(* Logix 5000 project; controller PBS_Perfusion vendor 1 type 14 code 217 rev 32.14; software revision 32.03; part 17 of 27 *)
(* tags used below, declared in another part *)
   P_Intlk : BOOL;   // Unique Parameter Name for auto - discovery
   REAL : DINT;
(* P_Intlk, continued *)

ROUTINE Prescan   (* ladder *)
// Clear "lurking" Commands
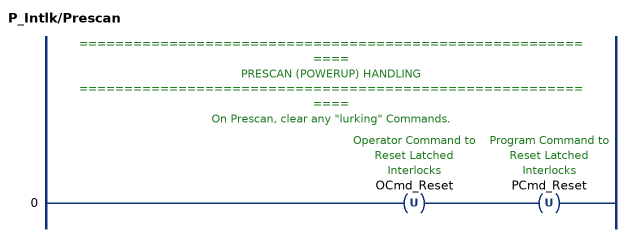
   // ============================================================
   // PRESCAN (POWERUP) HANDLING
   // ============================================================
   // On Prescan, clear any "lurking" Commands.
   0: OTU(OCmd_Reset)OTU(PCmd_Reset);
END_ROUTINE
END_ADD_ON_INSTRUCTION

ADD_ON_INSTRUCTION P_ValveC   (* revision 4.10 .01 Release, vendor Rockwell Automation, ExecutePrescan, ExecuteEnableInFalse *)
// Revision note:
// See Instruction Help for a summary of changes, and see 4.10 Release Notes for details.
// Help:
// Copyright © Rockwell Automation, Inc.  All Rights Reserved.
// This Instruction controls an Analog or Pulse Output Valve with
// analog or simulated position feedback and provides:
// *  Program and Operator entry of target position in Percent Open
// *  Ramping of position to target at specified Rate of Change (%/sec)
// *  Scaling of Position Feedback input from Raw (I/O card) Units to percent
// *  Monitoring of Interlock conditions which cause output to shed
// *  Configurable shed to HOLD or to configured position
// *  Monitoring of I/O communication faults
// *  Alarms for Interlock Trip, Actuator Fault, I/O Fault
// *  Operation in Hand, Maintenance, Override, Program and Operator Modes
// *  "Available" status for use by automation logic to know whether valve
//       can be controlled by other objects.
// Command Sources are arbitrated by a P_CmdSrc Add-On Instruction instance.
// Alarms are provided by P_Alarm Add-On Instruction instances.
// Command Sources: Operator, Program, External, Override, Maintenance, Out of Service, Hand
// Configuration notes:
//    If Max ON Time is less than 0 or greater than the Cycle Time
//         it is set to the Cycle Time.
//    If Min ON Time is less than 0 or greater than the Max ON Time
//         it is set to zero.
//    If Deadtime is less than 0 or greater than the Cycle Time,
//         it is set to zero.
//    Bump Time must be within the Min ON Time and Max ON Time.
// SUMMARY OF CHANGES FROM PREVIOUS VERSION (4.10.00)
// See 4.10 Release Notes for details.
// * No changes, uprevved because P_CmdSrc 4.10.01 is used.
// SUMMARY OF CHANGES FROM PREVIOUS VERSION (4.00.00)
// See 4.10 Release Notes for details.
// * Added option to clamp to a full/empty range when we have limit switches.
// * Changed availability to use input availability from interlocks.
// * Updated to P_CmdSrc V4.10.00.
// * Corrected parameter External Access.
// * Added Cfg_HasMoreObj.
// SUMMARY OF CHANGES FROM PREVIOUS VERSION (3.5-11)
// See 4.00 Release Notes for details.
// * Changed Inf_ items to HMI_, and added Cfg_Area for security.
// * Added notify and unack count rollup for associated object(s).
// * Changed "Mode" to "Command Source" using P_CmdSrc 4.00.00.
// * Deleted Cfg_PCmdClear; all Program Commands are now self-clearing.
// * Aligned ready bit naming with command bit names.
// * Added unacked alarm count.
// * Added  configurable decimal places for display on HMI.
// * All OCmds/MCmds and ORdys/MRdys are now Local Tags.
// * Added Sts_RdyAck and Sts_RdyReset for use by external objects.
// * Added option for no position feedback (simulated with hysteresis).
VAR_INPUT
   Inp_PosFdbk : REAL; {visible}   // Position Feedback from Valve (in Raw Input units)
   Inp_OpenLS : BOOL; {visible}   // Valve Open Limit Switch 1=confirmed fully open
   Inp_ClosedLS : BOOL; {visible}   // Valve Closed Limit Switch 1=confirmed fully closed
   Inp_ActuatorFault : BOOL; {visible}   // Valve Actuator Fault (overload, etc.), 0=OK, 1=Fault)
   Inp_IntlkOK : BOOL := 1; {visible}   // 1=Interlocks OK, Pulse Output Valve can be moved
   Inp_NBIntlkOK : BOOL := 1; {visible}   // 1=Non-Bypassable Interlocks OK, Pulse Output Valve can be moved
   Inp_IntlkAvail : BOOL;   // 1 = Interlock Availibility OK
   Inp_IOFault : BOOL;   // Input / Output Communication Status 0=OK, 1=fail
   Inp_Sim : BOOL;   // 1=I/O are being simulated, set output CV to 0.0, ignore I/O Fault
   Inp_Hand : ALIAS FOR CmdSrc.Inp_Hand;
   Inp_Ovrd : ALIAS FOR CmdSrc.Inp_Ovrd;
   Inp_OvrdCV : REAL;   // CV target in Override Mode (CV EU)
   Inp_ExtInh : ALIAS FOR CmdSrc.Inp_ExtInh;
   Inp_Reset : BOOL;   // 1=Reset shed latches and cleared alarms
   Cfg_ShedHold : BOOL;   // 1=Hold Output on Interlock or bad PV, 0=Go to Cfg_IntlkCV
   Cfg_ShedOnIOFault : BOOL := 1;   // 1=Take shed action (hold or interlock CV) on I/O Fault
   Cfg_SkipRoCLim : BOOL;   // 1=Skip RoC Limiting in Intlk, Maint, Ovrd modes
   Cfg_SetTrack : BOOL := 1;   // 1=PSets track OSets in Oper, OSets track PSets in Prog, 0=no tracking
   Cfg_SetTrackOvrdHand : BOOL;   // 1=Prog/Oper Settings track Override/Hand CV
   Cfg_HasPosFdbk : BOOL := 1;   // 1=Valve provides an analog position feedback, 0=simulate feedback
   Cfg_HasOpenLS : BOOL;   // 1=Valve provides an Open Limit Switch signal
   Cfg_HasClosedLS : BOOL;   // 1=Valve provides a Closed Limit Switch signal
   Cfg_UseOpenLS : BOOL;   // 1=Valve Open LS should be used for open/closed status
   Cfg_UseClosedLS : BOOL;   // 1=Valve Closed LS should be used for open/closed status
   Cfg_LSFail : BOOL := 1;   // 1=both switches ON=fail, 0=both switches OFF=fail
   Cfg_ClampPosToLS : BOOL;   // 1=Clamps Val_Pos to EUMin/Max when on a Limit Switch
   Cfg_HasIntlkObj : BOOL;   // 1=Tells HMI a P_Intlk is connected to Inp_Intlk
   Cfg_HasMoreObj : BOOL;   // 1=Tells HMI an object with more info is available
   Cfg_HasCVNav : BOOL;   // 1=Tells HMI to enable navigation to a connected CV object
   Cfg_OvrdIntlk : BOOL;   // 1=Override ignores Bypassable Intlk; 0=always use Intlk
   Cfg_DecPlcs : DINT;   // Number of decimal places for CV display (0..6)
   Cfg_HasIntlkTripAlm : ALIAS FOR IntlkTrip.Cfg_Exists;   // 1=Interlock Trip Alarm exists and will be checked
   Cfg_HasActuatorFaultAlm : ALIAS FOR ActuatorFault.Cfg_Exists;   // 1=Actuator Fault Alarm exists and will be checked
   Cfg_HasIOFaultAlm : ALIAS FOR IOFault.Cfg_Exists;   // 1=I/O Fault Alarm exists and will be checked
   Cfg_IntlkTripResetReqd : ALIAS FOR IntlkTrip.Cfg_ResetReqd;   // 1=Reset required to clear Interlock Trip Alarm
   Cfg_ActuatorFaultResetReqd : ALIAS FOR ActuatorFault.Cfg_ResetReqd;   // 1=Reset required to clear Actuator Fault Alarm
   Cfg_IOFaultResetReqd : ALIAS FOR IOFault.Cfg_ResetReqd;   // 1=Reset required to clear I/O Fault Alarm
   Cfg_IntlkTripAckReqd : ALIAS FOR IntlkTrip.Cfg_AckReqd;   // 1=Acknowledge required for Interlock Trip Alarm
   Cfg_ActuatorFaultAckReqd : ALIAS FOR ActuatorFault.Cfg_AckReqd;   // 1=Acknowledge required for Actuator Fault Alarm
   Cfg_IOFaultAckReqd : ALIAS FOR IOFault.Cfg_AckReqd;   // 1=Acknowledge required for I/O Fault Alarm
   Cfg_IntlkTripSeverity : ALIAS FOR IntlkTrip.Cfg_Severity;   // Interlock Trip Alarm Severity: 1..250=Low, 251..500=Medium, 501..750=High, 751..1000=Urgent
   Cfg_ActuatorFaultSeverity : ALIAS FOR ActuatorFault.Cfg_Severity;   // Actuator Fault Alarm Severity: 1..250=Low, 251..500=Medium, 501..750=High, 751..1000=Urgent
   Cfg_IOFaultSeverity : ALIAS FOR IOFault.Cfg_Severity;   // I/O Fault Alarm Severity: 1..250=Low, 251..500=Medium, 501..750=High, 751..1000=Urgent
   Cfg_MinCV : REAL;   // Minimum CV (in CV EU, for limiting)
   Cfg_MaxCV : REAL := 100.0;   // Maximum CV (in CV EU, for limiting)
   Cfg_CVRoCLimInc : REAL;   // CV Rate of Change Limit, Increasing, (EU/sec, 0=unlimited)
   Cfg_CVRoCLimDec : REAL;   // CV Rate of Change Limit, Decreasing, (EU/sec, 0=unlimited)
   Cfg_IntlkCV : REAL;   // CV (target in EU) when interlocked (if not Cfg_ShedHold)
   Cfg_CVEUMin : REAL;   // CV Minimum in Engineering Units (for scaling)
   Cfg_CVEUMax : REAL := 100.0;   // CV Maximum in Engineering Units (for scaling)
   Cfg_CVRawMin : REAL;   // CV Minimum in I/O (raw) Units (for scaling)
   Cfg_CVRawMax : REAL := 100.0;   // CV Maximum in I/O (raw) Units (for scaling)
   Cfg_FdbkRawMin : REAL;   // Position Feedback Minimum in raw input units (for scaling)
   Cfg_FdbkRawMax : REAL := 100.0;   // Position Feedback Maximum in raw input units (for scaling)
   Cfg_CycleT : REAL := 10.0;   // Open and Close Pulse Output overall period (s)
   Cfg_OpenRate : REAL := 1.0;   // Rate at which valve moves when opening (CV EU/sec)
   Cfg_CloseRate : REAL := 1.0;   // Rate at which valve moves when closing (CV EU/sec)
   Cfg_MaxOnT : REAL := 5.0;   // Open and Close Pulse Output maximum ON time (s)
   Cfg_MinOnT : REAL := 1.0;   // Open and Close Pulse Output minimum ON time (s)
   Cfg_BumpT : REAL;   // Time to bump valve open or closed (by Oper) when Fdbk Bad (sec)
   Cfg_Deadtime : REAL;   // Additional time on first pulse after stop or direction change
   Cfg_MaxClosedPos : REAL;   // Position above which valve is assumed open if limit switches not used
   PSet_CV : REAL;   // Program Setting of Controlled Variable (output) (CV EU)
   PSet_Owner : DINT;   // Program Owner Request ID (non-zero) or Release (zero)
   XSet_CV : REAL;   // External Setting of Controlled Variable (output) (CV EU)
   PCmd_Prog : ALIAS FOR CmdSrc.PCmd_Prog;
   PCmd_Oper : ALIAS FOR CmdSrc.PCmd_Oper;
   PCmd_Lock : ALIAS FOR CmdSrc.PCmd_Lock;
   PCmd_Unlock : ALIAS FOR CmdSrc.PCmd_Unlock;
   PCmd_Normal : ALIAS FOR CmdSrc.PCmd_Normal;
   PCmd_Reset : BOOL;   // Program Command to reset shed latches and cleared alarms
   PCmd_IntlkTripAck : ALIAS FOR IntlkTrip.PCmd_Ack;   // Program Command to Acknowledge Interlock Trip Alarm
   PCmd_IntlkTripSuppress : ALIAS FOR IntlkTrip.PCmd_Suppress;   // Program Command to Suppress Interlock Trip Alarm
   PCmd_IntlkTripUnsuppress : ALIAS FOR IntlkTrip.PCmd_Unsuppress;   // Program Command to Unsuppress Interlock Trip Alarm
   PCmd_IntlkTripUnshelve : ALIAS FOR IntlkTrip.PCmd_Unshelve;   // Program Command to Unshelve Interlock Trip Alarm
   PCmd_ActuatorFaultAck : ALIAS FOR ActuatorFault.PCmd_Ack;   // Program Command to Acknowledge Actuator Fault Alarm
   PCmd_ActuatorFaultSuppress : ALIAS FOR ActuatorFault.PCmd_Suppress;   // Program Command to Suppress Actuator Fault Alarm
   PCmd_ActuatorFaultUnsuppress : ALIAS FOR ActuatorFault.PCmd_Unsuppress;   // Program Command to Unsuppress Actuator Fault Alarm
   PCmd_ActuatorFaultUnshelve : ALIAS FOR ActuatorFault.PCmd_Unshelve;   // Program Command to Unshelve Actuator Fault Alarm
   PCmd_IOFaultAck : ALIAS FOR IOFault.PCmd_Ack;   // Program Command to Acknowledge I/O Fault Alarm
   PCmd_IOFaultSuppress : ALIAS FOR IOFault.PCmd_Suppress;   // Program Command to Suppress I/O Fault Alarm
   PCmd_IOFaultUnsuppress : ALIAS FOR IOFault.PCmd_Unsuppress;   // Program Command to Unsuppress I/O Fault Alarm
   PCmd_IOFaultUnshelve : ALIAS FOR IOFault.PCmd_Unshelve;   // Program Command to Unshelve I/O Fault Alarm
   MCmd_Rel : ALIAS FOR CmdSrc.MCmd_Rel;
   OCmd_Unlock : ALIAS FOR CmdSrc.OCmd_Unlock;
   XCmd_Acq : ALIAS FOR CmdSrc.XCmd_Acq;
   XCmd_Rel : ALIAS FOR CmdSrc.XCmd_Rel;
   XCmd_Reset : BOOL;   // External Command to reset shed latches and cleared alarms
END_VAR
VAR_OUTPUT
   Out_CV : REAL; {access Read Only, visible}   // CV Output in Raw (I/O Card) Units
   Out_Open : BOOL; {access Read Only, visible}   // Pulse Output to drive valve Open
   Out_Close : BOOL; {access Read Only, visible}   // Pulse Output to drive valve closed
   Val_Pos : REAL; {access Read Only, visible}   // Valve actual position from feedback (CV EU)
   Val_CVSet : REAL; {access Read Only, visible}   // Value of selected CV Setting (before rate limiting, CV EU)
   Val_CVOut : REAL; {access Read Only, visible}   // Value of CV output (after clamping and ramping) (CV EU)
   Val_CVEUMin : REAL; {access Read Only}   // Minimum of scaled range = MIN (Cfg_CVEUMin, Cfg_CVEUMax)
   Val_CVEUMax : REAL := 100.0; {access Read Only}   // Maximum of scaled range = MAX (Cfg_CVEUMin, Cfg_CVEUMax)
   SrcQ_IO : DINT; {access Read Only}   // Source and Quality of primary I/O (enumeration)
   SrcQ : DINT; {access Read Only}   // Source and Quality of primary Val/Sts (enumeration)
   Val_Fdbk : DINT; {access Read Only}   // Device Feedback 0=Moving, 1=Closed, 2=Opened, 3=Limit Switch Failure
   Val_Sts : DINT; {access Read Only}   // 0=AtTarget, 1=RampClose, 2=RampOpen, 3=Clamp@Min, 4=Clamp@Max, 5=BumpClose, 6=BumpOpen
   Val_Fault : DINT; {access Read Only}   // Device Fault Status 0=none, 32=I/OFault, 34=CfgErr
   Val_NotifyAll : DINT; {access Read Only}   // Highest Alarm prio and ack status this object + channel (enum)
   Val_UnackAlmC : DINT; {access Read Only}   // Count of Unacknowledged Alarms
   Val_Owner : DINT; {access Read Only}   // Current Object Owner ID (0=not owned)
   Sts_CVInfNaN : BOOL; {access Read Only}   // 1=Selected CV is Infinite or Not A Number (1.$, 1.#NaN)
   Sts_PosInfNaN : BOOL; {access Read Only}   // 1=Inp_PosFdbk is Infinite or Not A Number (1.$, 1.#NaN)
   Sts_BumpOpen : BOOL; {access Read Only}   // 1=Bump Open Requested or Active
   Sts_BumpClose : BOOL; {access Read Only}   // 1=Bump Close Requested or Active
   Sts_Ramping : BOOL; {access Read Only}   // 1=CV is ramping to target
   Sts_Clamped : BOOL; {access Read Only}   // 1=CV Set is clamped at CVMin or CVMax
   Sts_SkipRoCLim : BOOL; {access Read Only}   // 1=Rate of Change Limiting was skipped this scan (Maint, Ovrd, Intlk, Hand)
   Sts_Active : BOOL; {access Read Only}   // 1=CV is greater than Cfg_MaxClosedPos, show valve symbol as "opened"
   Sts_Available : BOOL; {access Read Only}   // 1=Pulse Output Valve available for control by automation (Prog)
   Sts_Bypass : BOOL; {access Read Only}   // 1=Bypassable Interlocks are Bypassed
   Sts_BypActive : BOOL; {access Read Only}   // 1=Bypassing Active (Bypassed or Maintenance)
   Sts_LSFail : BOOL; {access Read Only}   // 1=Limit Switch Overlap Failure
   Sts_NotRdy : BOOL; {access Read Only}   // 1=Device Not Ready, see detail bits for reason
   Nrdy_CfgErr : BOOL; {access Read Only}   // 1=Device Not Ready: Configuration Error
   Nrdy_Intlk : BOOL; {access Read Only}   // 1=Device Not Ready: Interlock Not OK
   Nrdy_IOFault : BOOL; {access Read Only}   // 1=Device Not Ready: I/O Fault (Shed Requires Reset)
   Nrdy_OoS : BOOL; {access Read Only}   // 1=Device Not Ready: Device is Out of Service
   Sts_MaintByp : BOOL; {access Read Only}   // 1=Device has a Maintenance Bypass function active
   Sts_AlmInh : BOOL; {access Read Only}   // 1=One or more Alarms Shelved, Disabled or Suppressed
   Sts_Err : BOOL; {access Read Only, visible}   // 1=Error in Config: see detail bits for reason
   Err_Limit : BOOL; {access Read Only}   // 1=Error in Config: CV Limits swapped
   Err_EU : BOOL; {access Read Only}   // 1=Error in Config: Scaled CV EU Min = Max
   Err_Raw : BOOL; {access Read Only}   // 1=Error in Config: Raw Output Scaling Min = Max
   Err_Fdbk : BOOL; {access Read Only}   // 1=Error in Config: Raw Feedback Scaling Min = Max
   Err_Timer : BOOL; {access Read Only}   // 1=Error in Config: Invalid Timer Preset (use 0 to 2147483)
   Err_Alarm : BOOL; {access Read Only}   // 1=Error in Config: Alarm Min On Time, Shelf Time, Severity
   Sts_Hand : ALIAS FOR CmdSrc.Sts_Hand; {access Read Only, visible}
   Sts_OoS : ALIAS FOR CmdSrc.Sts_OoS; {access Read Only, visible}
   Sts_Maint : ALIAS FOR CmdSrc.Sts_Maint; {access Read Only, visible}
   Sts_Ovrd : ALIAS FOR CmdSrc.Sts_Ovrd; {access Read Only, visible}
   Sts_Ext : ALIAS FOR CmdSrc.Sts_Ext; {access Read Only, visible}
   Sts_Prog : ALIAS FOR CmdSrc.Sts_Prog; {access Read Only, visible}
   Sts_ProgLocked : ALIAS FOR CmdSrc.Sts_ProgLocked; {access Read Only}
   Sts_Oper : ALIAS FOR CmdSrc.Sts_Oper; {access Read Only, visible}
   Sts_OperLocked : ALIAS FOR CmdSrc.Sts_OperLocked; {access Read Only}
   Sts_Normal : ALIAS FOR CmdSrc.Sts_Normal; {access Read Only}
   Sts_ExtReqInh : ALIAS FOR CmdSrc.Sts_ExtReqInh; {access Read Only}
   Sts_ProgReqInh : ALIAS FOR CmdSrc.Sts_ProgReqInh; {access Read Only}
   Sts_MAcqRcvd : ALIAS FOR CmdSrc.Sts_MAcqRcvd; {access Read Only}
   Sts_RdyReset : ALIAS FOR ORdy_Reset; {access Read Only}   // 1=A latched alarm or shed condition is ready to be reset
   Sts_RdyAck : BOOL; {access Read Only}   // 1=An alarm is ready to be acknowledged
   Sts_IntlkTrip : ALIAS FOR IntlkTrip.Inp;   // 1=Status: CV held or forced by interlock NOT OK (1-shot)
   Alm_IntlkTrip : ALIAS FOR IntlkTrip.Alm;   // 1=Alarm: CV held or forced by interlock NOT OK
   Ack_IntlkTrip : ALIAS FOR IntlkTrip.Ack;   // 1=Interlock Trip Alarm has been acknowledged
   Sts_IntlkTripDisabled : ALIAS FOR IntlkTrip.Disabled;   // 1=Interlock Trip Alarm has been Disabled by Maintenance
   Sts_IntlkTripShelved : ALIAS FOR IntlkTrip.Shelved;   // 1=Interlock Trip Alarm has been Shelved by Operator
   Sts_IntlkTripSuppressed : ALIAS FOR IntlkTrip.Suppressed;   // 1=Interlock Trip Alarm has been Suppressed by Program
   Sts_ActuatorFault : ALIAS FOR ActuatorFault.Inp;   // 1=Actuator Fault detected (input)
   Alm_ActuatorFault : ALIAS FOR ActuatorFault.Alm;   // 1=Alarm: Actuator Fault Detected
   Ack_ActuatorFault : ALIAS FOR ActuatorFault.Ack;   // 1=Actuator Fault Alarm has been acknowledged
   Sts_ActuatorFaultDisabled : ALIAS FOR ActuatorFault.Disabled;   // 1=Actuator Fault Alarm has been Disabled by Maintenance
   Sts_ActuatorFaultShelved : ALIAS FOR ActuatorFault.Shelved;   // 1=Actuator Fault Alarm has been Shelved by Operator
   Sts_ActuatorFaultSuppressed : ALIAS FOR ActuatorFault.Suppressed;   // 1=Actuator Fault Alarm has been Suppressed by Program
   Sts_IOFault : ALIAS FOR IOFault.Inp;   // 1=I/O Fault Status (0=OK, 1=Bad)
   Alm_IOFault : ALIAS FOR IOFault.Alm;   // 1=I/O Fault Alarm
   Ack_IOFault : ALIAS FOR IOFault.Ack;   // 1=I/O Fault Alarm has been acknowledged
   Sts_IOFaultDisabled : ALIAS FOR IOFault.Disabled;   // 1=I/O Fault Alarm has been Disabled by Maintenance
   Sts_IOFaultShelved : ALIAS FOR IOFault.Shelved;   // 1=I/O Fault Alarm has been Shelved by Operator
   Sts_IOFaultSuppressed : ALIAS FOR IOFault.Suppressed;   // 1=I/O Fault Alarm has been Suppressed by Program
   MRdy_Rel : ALIAS FOR CmdSrc.MRdy_Rel; {access Read Only}
   ORdy_Unlock : ALIAS FOR CmdSrc.ORdy_Unlock; {access Read Only}
   P_ValveC : BOOL;   // Unique Parameter Name for auto - discovery
END_VAR
VAR
   CmdSrc : P_CmdSrc := (Cfg_HasOper := 1, Cfg_HasOperLocked := 1, Cfg_HasProg := 1, Cfg_HasProgLocked := 1, Cfg_HasMaint := 1, Cfg_HasMOoS := 1, Cfg_OvrdOverLock := 1, Sts_bSrc := 1);   // Control / Command Source Selection
   IOFault : P_Alarm := (Cfg_AckReqd := 1, Cfg_AllowShelve := 1, Cfg_AllowDisable := 1, Cfg_Severity := 1000, Cfg_AlmMinOnT := 5, PCfg_AllowExist := 1, Ack := 1);   // I/O Fault Alarm
   IntlkTrip : P_Alarm := (Cfg_AckReqd := 1, Cfg_AllowShelve := 1, Cfg_AllowDisable := 1, Cfg_Severity := 500, Cfg_AlmMinOnT := 5, PCfg_AllowExist := 1, Ack := 1);   // Interlock Trip Alarm
   Cfg_Tag : STRING_20 := 'P_ValveC';   // Tagname for display on HMI
   Cfg_Label : STRING_20 := 'Control Valve';   // Label for graphic symbol displayed on HMI
   Cfg_Desc : STRING_40 := 'Control Valve';   // Description for display on HMI
   Wrk_Notify : DINT; {access None}   // Buffer for building Val_Notify
   Wrk_Bypass : BOOL; {access None}   // Internal Bypassable Interlocks are Bypassed flag
   Cfg_EU : STRING_8 := '% Open';   // Engineering Units for display on HMI
   Wrk_CV : REAL; {access None}   // Working copy of Speed Reference (for limiting)
   Wrk_CVSet : REAL; {access None}   // Final selected CV to feed to RoC Limiter
   Wrk_CVOut : REAL; {access None}   // Working value of CV after Rate Limiting
   Wrk_IntlkTripONS : BOOL; {access None}   // Interlock Tripped This Scan
   Wrk_ScanTime : REAL; {access None}   // Seconds since previous scan
   Wrk_StepInc : REAL; {access None}   // Amount to increase CV (to valve pulse logic) this scan for rate limiting
   Wrk_ScanT : TIMER := (PRE := 2147483647); {access None}   // Scan Timer (milliseconds, always runs)
   HMI_Tab : SINT;   // Tab to display (FTView ME)
   Wrk_Sts : DINT; {access None}   // Buffer for building Val_Sts
   Wrk_Fault : DINT; {access None}   // Buffer for building Val_Fault
   Wrk_SrcQ : DINT; {access None}   // Register for building Source / Quality enumeration
   ActuatorFault : P_Alarm := (Cfg_AckReqd := 1, Cfg_AllowShelve := 1, Cfg_AllowDisable := 1, Cfg_Severity := 1000, Cfg_AlmMinOnT := 5, PCfg_AllowExist := 1, Ack := 1);   // Actuator Fault Alarm (based on Actuator Fault Input)
   Wrk_RealChkDINT : DINT; {access None}   // REAL tag bit pattern as a DINT to check for Inf / NaN
   Wrk_Close : BOOL; {access None}   // Internal Close output -- before Sim
   Wrk_Open : BOOL; {access None}   // Internal Open output -- before Sim
   Wrk_CycleT : TIMER := (PRE := 2147483647); {access None}   // Overall Cycle Timer for pulsed outputs
   Wrk_OKtoOpen : BOOL; {access None}   // OK to pulse Out_Open
   Wrk_OKtoClose : BOOL; {access None}   // OK to pulse Out_Close
   Wrk_OpenTime : REAL; {access None}   // Time to pulse Out_Open
   Wrk_CycleT_ms : DINT; {access None}   // Cycle Time in milliseconds (preset)
   Wrk_OpenTimePrev : DINT; {access None}   // Wrk_OpenTime from previous cycle
   Wrk_CloseTime : REAL; {access None}   // Time to pulse Out_Close
   Wrk_CloseTimePrev : REAL; {access None}   // Wrk_CloseTime from previous cycle
   HMI_Type : STRING_16 := 'P_ValveC'; {access Read Only}   // Must contain AOI name, used for HMI and Information S/W
   Wrk_OpenFdbk : BOOL; {access None}   // 1=LS Feedback shows valve confirmed open
   Wrk_ClosedFdbk : BOOL; {access None}   // 1=LS Feedback shows valve confirmed closed
   Wrk_StepDec : REAL; {access None}   // Amount to decrease CV (to valve pulse logic) this scan for rate limiting
   Wrk_BumpClose : BOOL; {access None}   // Operator Bump Close requested
   Wrk_BumpOpen : BOOL; {access None}   // Operator Bump Open requested
   Wrk_BumpingOpen : BOOL; {access None}   // Operator Bump Open actively pulsing Out_Open
   Wrk_BumpingClose : BOOL; {access None}   // Operator Bump Close actively pulsing Out_Close
   Wrk_CycleActive : BOOL; {access None}   // Outputs are cycling; wait for cycle to complete
   HMI_Lib : STRING_12 := 'RA-BAS'; {access Read Only}   // Display Library for Faceplate call-up
   Cfg_CVNavTag : STRING_NavTag;   // Tagname for destination of CV Navigation button
   Wrk_ShedIntlkCV : BOOL; {access None}   // Output CV being held at Interlock value
   Wrk_ShedHold : BOOL; {access None}   // Output CV being held at last good value
   Cfg_Area : STRING_Area := 'area01';   // Process Area for security
   OSet_CV : REAL;   // Operator Setting of Controlled Variable (output) (CV EU)
   OCmd_ResetAckAll : BOOL;   // Oper Cmd to reset shed latches and cleared alarms and acknowledge all alarms
   OCmd_Reset : BOOL;   // Oper Cmd to reset shed latches and cleared alarms
   MCmd_Check : BOOL;   // Maintenance Command to Check (not bypass) all Interlocks
   MCmd_Bypass : BOOL;   // Maintenance Command to Bypass all Bypassable Interlocks
   OCmd_BumpClose : BOOL;   // Operator Command to bump valve closed (avail. if Fdbk Bad)
   OCmd_BumpOpen : BOOL;   // Operator Command to bump valve open (avail. if Fdbk Bad)
   ORdy_CV : BOOL; {access Read Only}   // 1=Ready for OSet_CV (enables data entry field)
   ORdy_ResetAckAll : BOOL; {access Read Only}   // 1=Ready for OCmd_ResetAckAll (enables HMI button)
   ORdy_Reset : BOOL; {access Read Only}   // 1=Ready for OCmd_Reset (enables HMI button)
   MRdy_Check : BOOL; {access Read Only}   // 1=Ready for MCmd_Check (enables HMI button)
   MRdy_Bypass : BOOL; {access Read Only}   // 1=Ready for MCmd_Bypass (enables HMI button)
   ORdy_BumpClose : BOOL; {access Read Only}   // 1=Ready for OCmd_BumpClose (enables HMI button)
   ORdy_BumpOpen : BOOL; {access Read Only}   // 1=Ready for OCmd_BumpOpen (enables HMI button)
   Wrk_UnackAlmC : DINT; {access None}   // Buffer for building Val_UnackAlmC
   Val_Notify : DINT; {access Read Only}   // Current Alarm Level and Acknowledgement (enumeration)
   Wrk_DeadtimeT : TIMER; {access None}   // Timer for valve hysteresis (deadtime)
   Wrk_LastMove : BOOL; {access None}   // 1=Last move was to open, 0=Last move was to close
   Wrk_WaitDeadtime : BOOL; {access None}   // 1=Need to wait deadtime before simulated move
END_VAR

ROUTINE EnableInFalse   (* ladder *)
// Out of Service is asserted, Output OFF (zero), Alarms inhibited
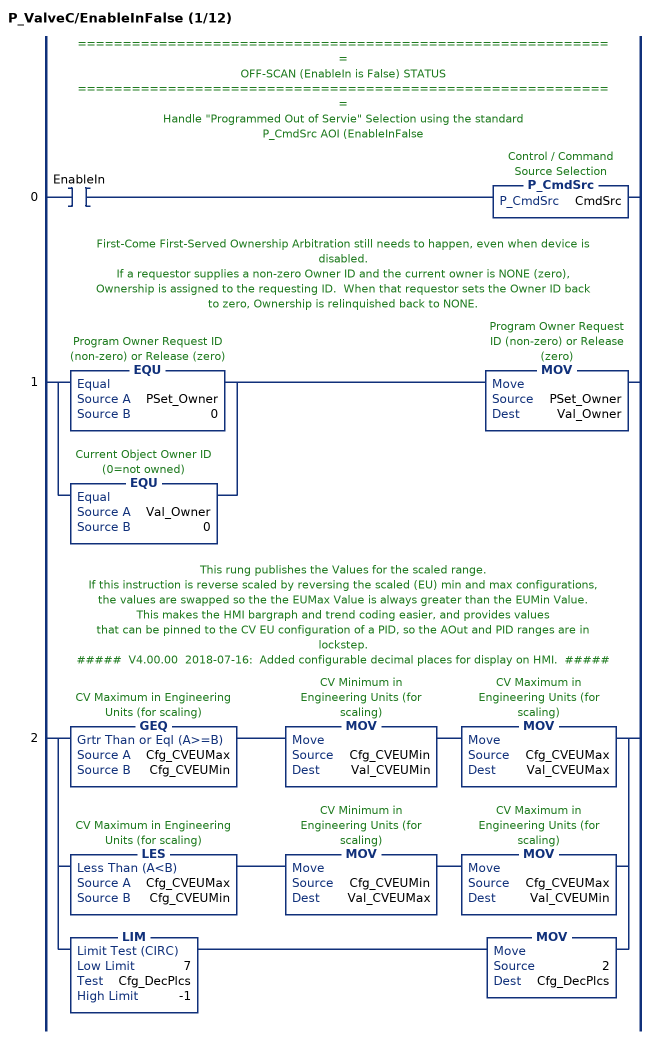
   // ============================================================
   // OFF-SCAN (EnableIn is False) STATUS
   // ============================================================
   // Handle "Programmed Out of Servie" Selection using the standard
   // P_CmdSrc AOI (EnableInFalse
   0: XIC(EnableIn)P_CmdSrc(CmdSrc);
   // First-Come First-Served Ownership Arbitration still needs to happen, even when device is disabled.
   // If a requestor supplies a non-zero Owner ID and the current owner is NONE (zero),
   // Ownership is assigned to the requesting ID.  When that requestor sets the Owner ID back
   // to zero, Ownership is relinquished back to NONE.
   1: [EQU(PSet_Owner,0) ,EQU(Val_Owner,0) ]MOV(PSet_Owner,Val_Owner);
   // This rung publishes the Values for the scaled range.
   // If this instruction is reverse scaled by reversing the scaled (EU) min and max configurations,
   // the values are swapped so the the EUMax Value is always greater than the EUMin Value.
   // This makes the HMI bargraph and trend coding easier, and provides values
   // that can be pinned to the CV EU configuration of a PID, so the AOut and PID ranges are in lockstep.
   // #####  V4.00.00  2018-07-16:  Added configurable decimal places for display on HMI.  #####
   2: [GEQ(Cfg_CVEUMax,Cfg_CVEUMin) MOV(Cfg_CVEUMin,Val_CVEUMin) MOV(Cfg_CVEUMax,Val_CVEUMax) ,LES(Cfg_CVEUMax,Cfg_CVEUMin) MOV(Cfg_CVEUMin,Val_CVEUMax) MOV(Cfg_CVEUMax,Val_CVEUMin) ,LIM(7,Cfg_DecPlcs,-1) MOV(2,Cfg_DecPlcs) ];
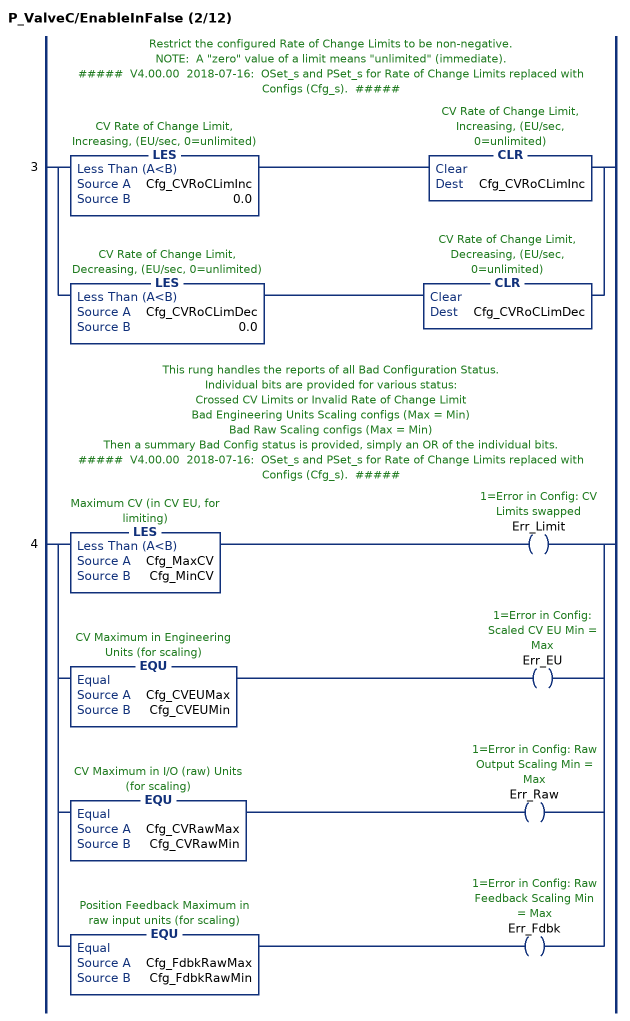
   // Restrict the configured Rate of Change Limits to be non-negative.
   // NOTE:  A "zero" value of a limit means "unlimited" (immediate).
   // #####  V4.00.00  2018-07-16:  OSet_s and PSet_s for Rate of Change Limits replaced with Configs (Cfg_s).  #####
   3: [LES(Cfg_CVRoCLimInc,0.0) CLR(Cfg_CVRoCLimInc) ,LES(Cfg_CVRoCLimDec,0.0) CLR(Cfg_CVRoCLimDec) ];
   // This rung handles the reports of all Bad Configuration Status.
   // Individual bits are provided for various status:
   // Crossed CV Limits or Invalid Rate of Change Limit
   // Bad Engineering Units Scaling configs (Max = Min)
   // Bad Raw Scaling configs (Max = Min)
   // Then a summary Bad Config status is provided, simply an OR of the individual bits.
   // #####  V4.00.00  2018-07-16:  OSet_s and PSet_s for Rate of Change Limits replaced with Configs (Cfg_s).  #####
   4: [LES(Cfg_MaxCV,Cfg_MinCV) OTE(Err_Limit) ,EQU(Cfg_CVEUMax,Cfg_CVEUMin) OTE(Err_EU) ,EQU(Cfg_CVRawMax,Cfg_CVRawMin) OTE(Err_Raw) ,EQU(Cfg_FdbkRawMax,Cfg_FdbkRawMin) OTE(Err_Fdbk) ];
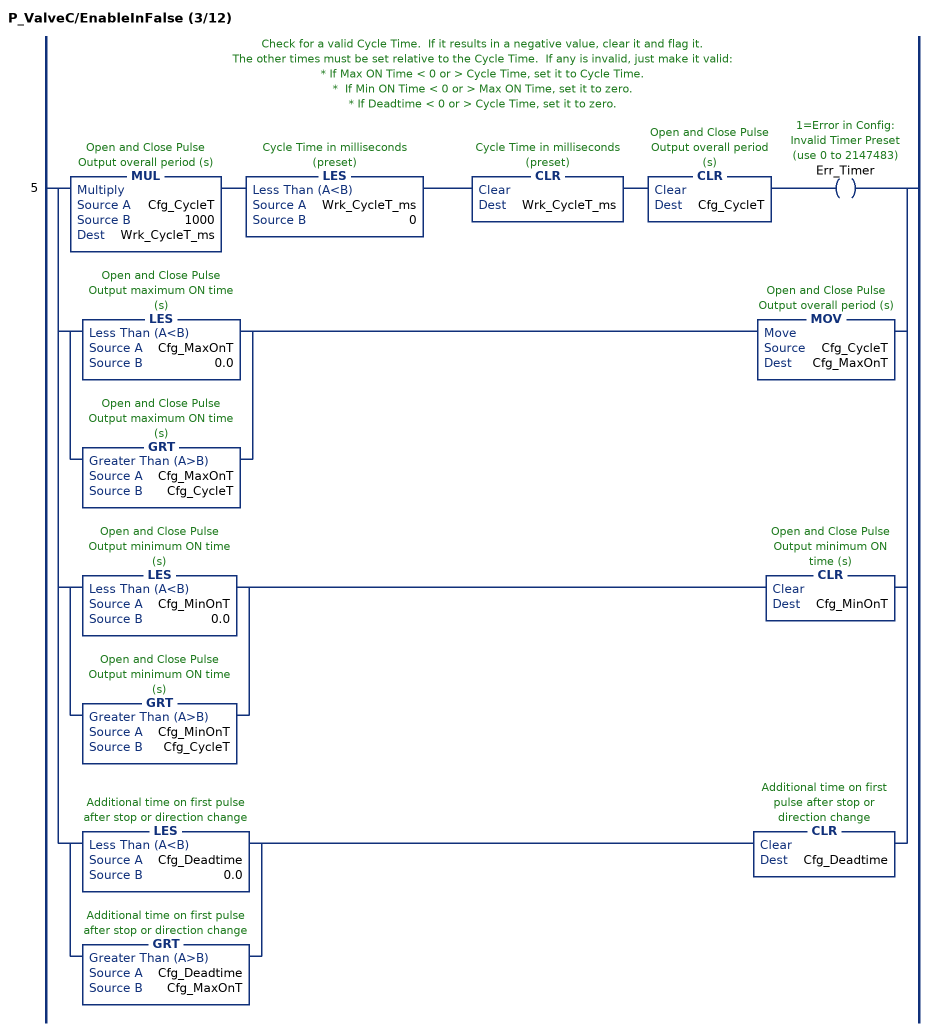
   // Check for a valid Cycle Time.  If it results in a negative value, clear it and flag it.
   // The other times must be set relative to the Cycle Time.  If any is invalid, just make it valid:
   // * If Max ON Time < 0 or > Cycle Time, set it to Cycle Time.
   // *  If Min ON Time < 0 or > Max ON Time, set it to zero.
   // * If Deadtime < 0 or > Cycle Time, set it to zero.
   5: [MUL(Cfg_CycleT,1000,Wrk_CycleT_ms) LES(Wrk_CycleT_ms,0) CLR(Wrk_CycleT_ms) CLR(Cfg_CycleT) OTE(Err_Timer) ,[LES(Cfg_MaxOnT,0.0) ,GRT(Cfg_MaxOnT,Cfg_CycleT) ] MOV(Cfg_CycleT,Cfg_MaxOnT) ,[LES(Cfg_MinOnT,0.0) ,GRT(Cfg_MinOnT,Cfg_CycleT) ] CLR(Cfg_MinOnT) ,[LES(Cfg_Deadtime,0.0) ,GRT(Cfg_Deadtime,Cfg_MaxOnT) ] CLR(Cfg_Deadtime) ];
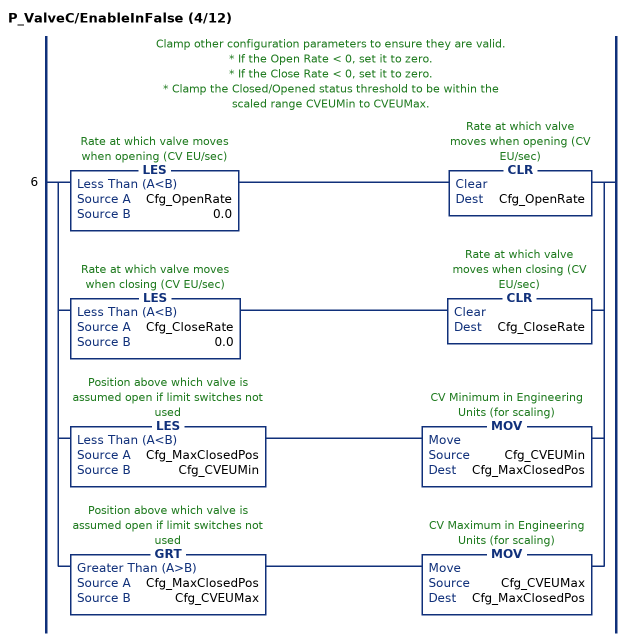
   // Clamp other configuration parameters to ensure they are valid.
   // * If the Open Rate < 0, set it to zero.
   // * If the Close Rate < 0, set it to zero.
   // * Clamp the Closed/Opened status threshold to be within the
   // scaled range CVEUMin to CVEUMax.
   6: [LES(Cfg_OpenRate,0.0) CLR(Cfg_OpenRate) ,LES(Cfg_CloseRate,0.0) CLR(Cfg_CloseRate) ,LES(Cfg_MaxClosedPos,Cfg_CVEUMin) MOV(Cfg_CVEUMin,Cfg_MaxClosedPos) ,GRT(Cfg_MaxClosedPos,Cfg_CVEUMax) MOV(Cfg_CVEUMax,Cfg_MaxClosedPos) ];
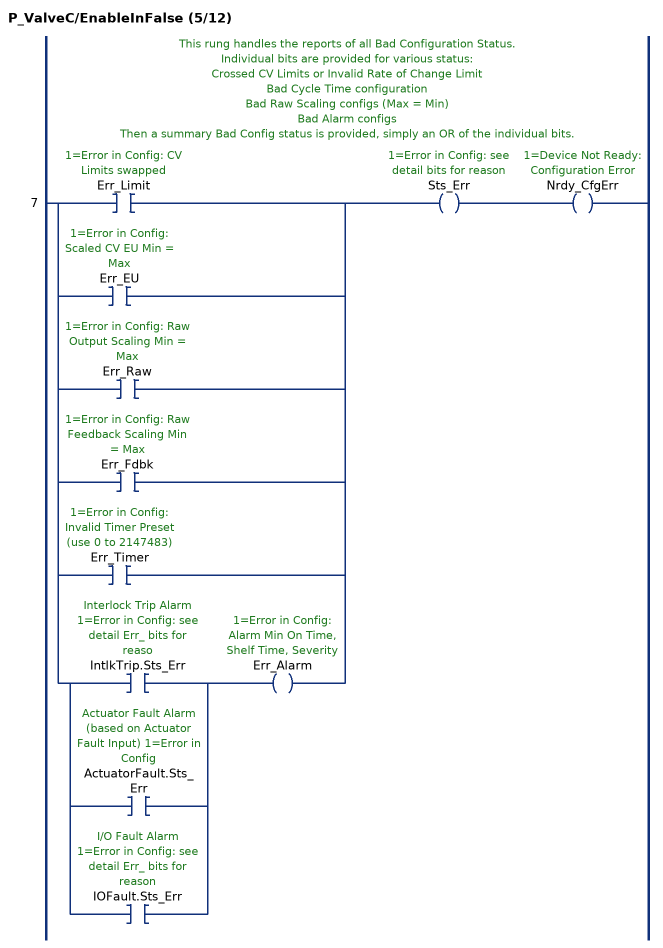
   // This rung handles the reports of all Bad Configuration Status.
   // Individual bits are provided for various status:
   // Crossed CV Limits or Invalid Rate of Change Limit
   // Bad Cycle Time configuration
   // Bad Raw Scaling configs (Max = Min)
   // Bad Alarm configs
   // Then a summary Bad Config status is provided, simply an OR of the individual bits.
   7: [XIC(Err_Limit) ,XIC(Err_EU) ,XIC(Err_Raw) ,XIC(Err_Fdbk) ,XIC(Err_Timer) ,[XIC(IntlkTrip.Sts_Err) ,XIC(ActuatorFault.Sts_Err) ,XIC(IOFault.Sts_Err) ] OTE(Err_Alarm) ]OTE(Sts_Err)OTE(Nrdy_CfgErr);
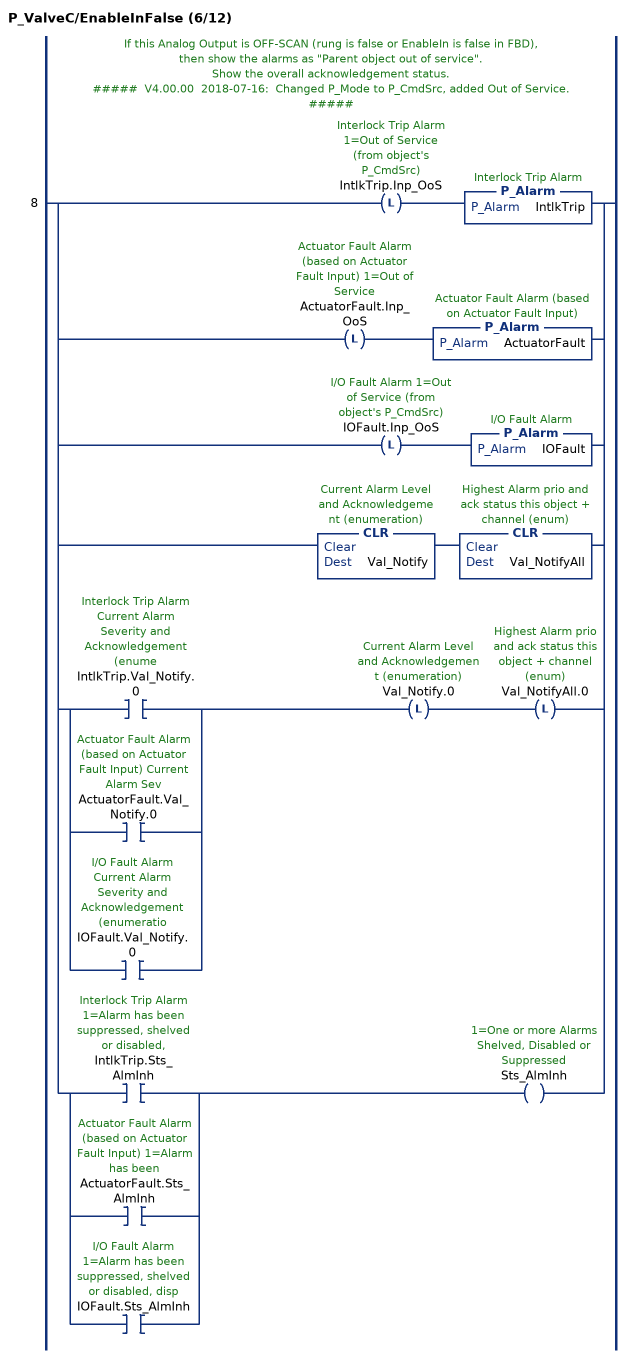
   // If this Analog Output is OFF-SCAN (rung is false or EnableIn is false in FBD),
   // then show the alarms as "Parent object out of service".
   // Show the overall acknowledgement status.
   // #####  V4.00.00  2018-07-16:  Changed P_Mode to P_CmdSrc, added Out of Service.  #####
   8: [OTL(IntlkTrip.Inp_OoS) P_Alarm(IntlkTrip) ,OTL(ActuatorFault.Inp_OoS) P_Alarm(ActuatorFault) ,OTL(IOFault.Inp_OoS) P_Alarm(IOFault) ,CLR(Val_Notify) CLR(Val_NotifyAll) ,[XIC(IntlkTrip.Val_Notify.0) ,XIC(ActuatorFault.Val_Notify.0) ,XIC(IOFault.Val_Notify.0) ] OTL(Val_Notify.0) OTL(Val_NotifyAll.0) ,[XIC(IntlkTrip.Sts_AlmInh) ,XIC(ActuatorFault.Sts_AlmInh) ,XIC(IOFault.Sts_AlmInh) ] OTE(Sts_AlmInh) ];
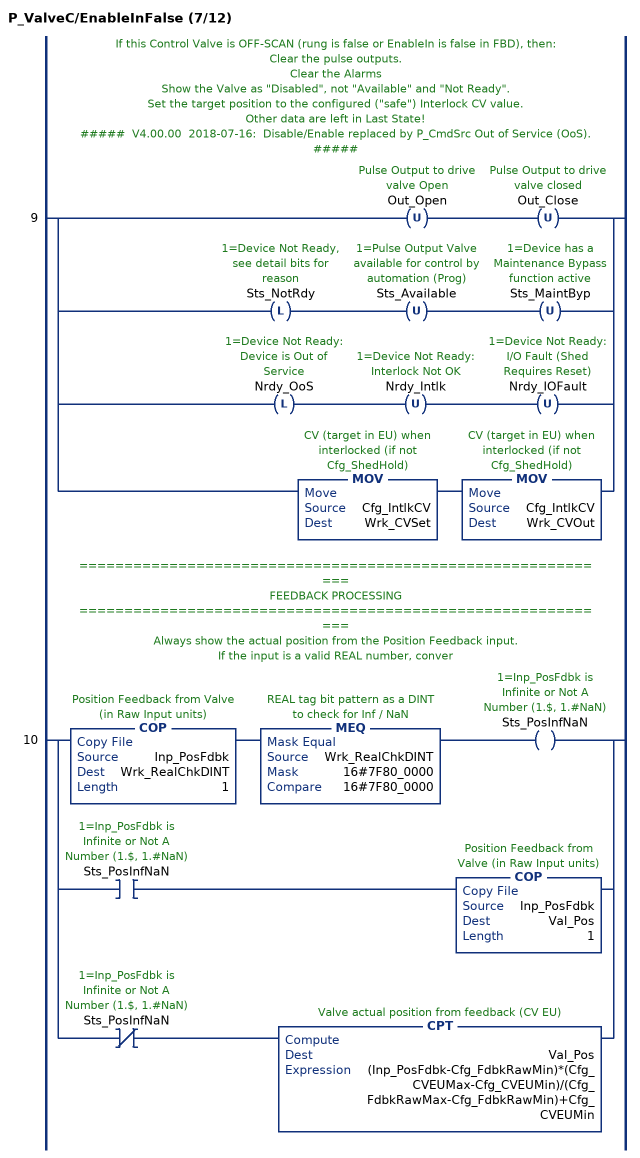
   // If this Control Valve is OFF-SCAN (rung is false or EnableIn is false in FBD), then:
   // Clear the pulse outputs.
   // Clear the Alarms
   // Show the Valve as "Disabled", not "Available" and "Not Ready".
   // Set the target position to the configured ("safe") Interlock CV value.
   // Other data are left in Last State!
   // #####  V4.00.00  2018-07-16:  Disable/Enable replaced by P_CmdSrc Out of Service (OoS).  #####
   9: [OTU(Out_Open) OTU(Out_Close) ,OTL(Sts_NotRdy) OTU(Sts_Available) OTU(Sts_MaintByp) ,OTL(Nrdy_OoS) OTU(Nrdy_Intlk) OTU(Nrdy_IOFault) ,MOV(Cfg_IntlkCV,Wrk_CVSet) MOV(Cfg_IntlkCV,Wrk_CVOut) ];
   // ============================================================
   // FEEDBACK PROCESSING
   // ============================================================
   // Always show the actual position from the Position Feedback input.
   // If the input is a valid REAL number, conver
   10: [COP(Inp_PosFdbk,Wrk_RealChkDINT,1) MEQ(Wrk_RealChkDINT,16#7F80_0000,16#7F80_0000) OTE(Sts_PosInfNaN) ,XIC(Sts_PosInfNaN) COP(Inp_PosFdbk,Val_Pos,1) ,XIO(Sts_PosInfNaN) CPT(Val_Pos,(Inp_PosFdbk-Cfg_FdbkRawMin)*(Cfg_CVEUMax-Cfg_CVEUMin)/(Cfg_FdbkRawMax-Cfg_FdbkRawMin)+Cfg_CVEUMin) ];
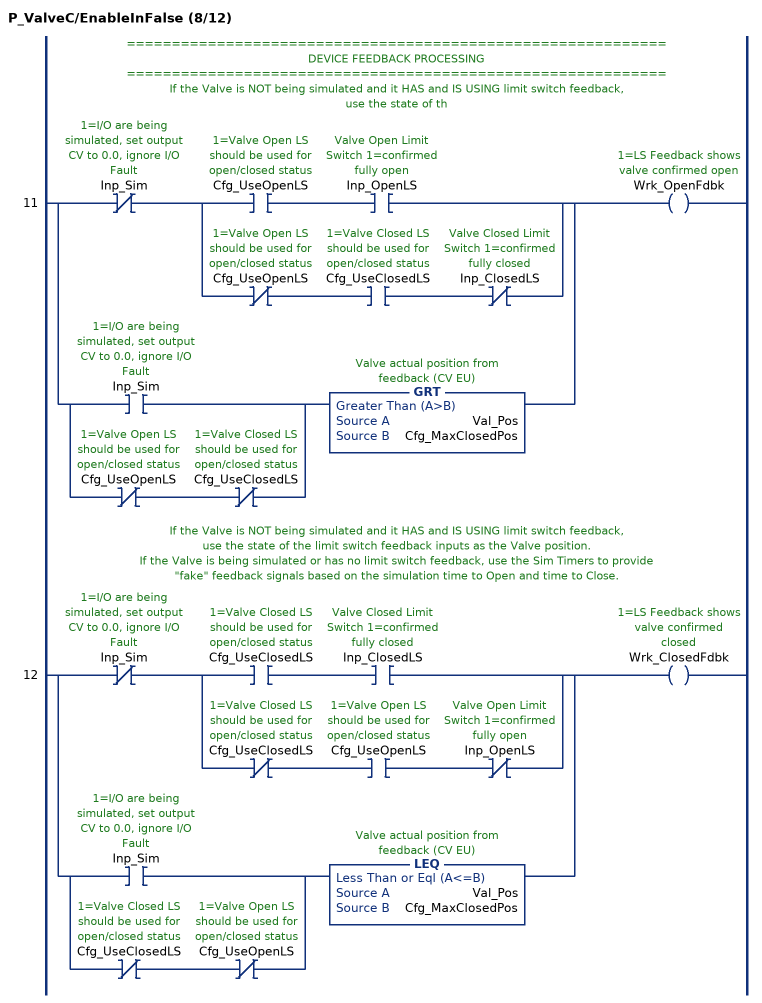
   // ============================================================
   // DEVICE FEEDBACK PROCESSING
   // ============================================================
   // If the Valve is NOT being simulated and it HAS and IS USING limit switch feedback,
   // use the state of th
   11: [XIO(Inp_Sim) [XIC(Cfg_UseOpenLS) XIC(Inp_OpenLS) ,XIO(Cfg_UseOpenLS) XIC(Cfg_UseClosedLS) XIO(Inp_ClosedLS) ] ,[XIC(Inp_Sim) ,XIO(Cfg_UseOpenLS) XIO(Cfg_UseClosedLS) ] GRT(Val_Pos,Cfg_MaxClosedPos) ]OTE(Wrk_OpenFdbk);
   // If the Valve is NOT being simulated and it HAS and IS USING limit switch feedback,
   // use the state of the limit switch feedback inputs as the Valve position.
   // If the Valve is being simulated or has no limit switch feedback, use the Sim Timers to provide
   // "fake" feedback signals based on the simulation time to Open and time to Close.
   12: [XIO(Inp_Sim) [XIC(Cfg_UseClosedLS) XIC(Inp_ClosedLS) ,XIO(Cfg_UseClosedLS) XIC(Cfg_UseOpenLS) XIO(Inp_OpenLS) ] ,[XIC(Inp_Sim) ,XIO(Cfg_UseClosedLS) XIO(Cfg_UseOpenLS) ] LEQ(Val_Pos,Cfg_MaxClosedPos) ]OTE(Wrk_ClosedFdbk);
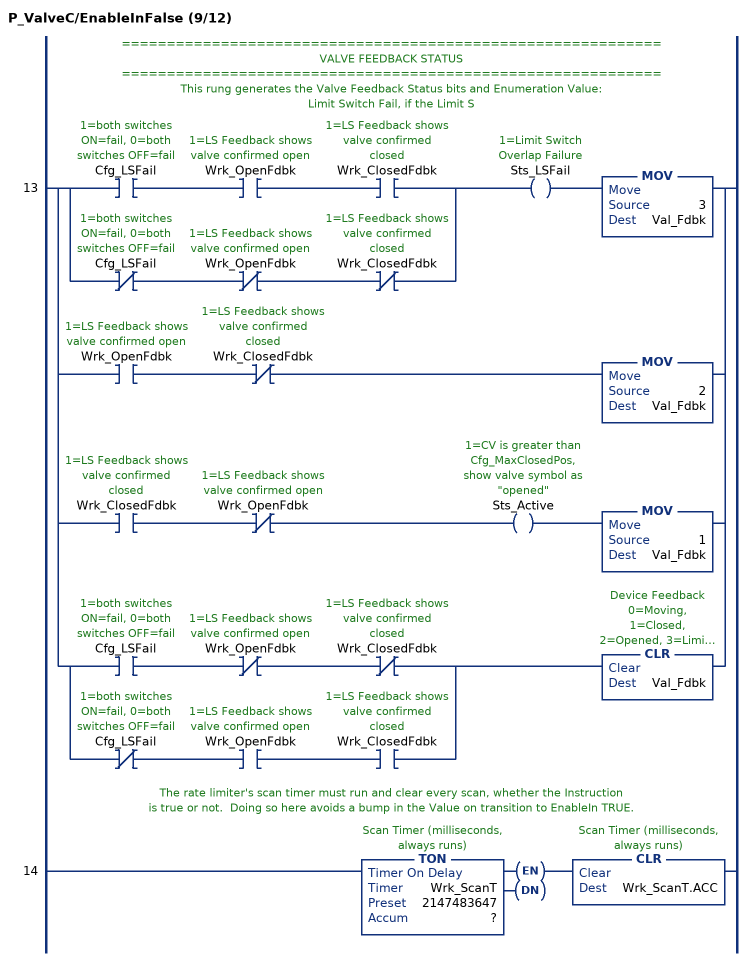
   // ============================================================
   // VALVE FEEDBACK STATUS
   // ============================================================
   // This rung generates the Valve Feedback Status bits and Enumeration Value:
   // Limit Switch Fail, if the Limit S
   13: [[XIC(Cfg_LSFail) XIC(Wrk_OpenFdbk) XIC(Wrk_ClosedFdbk) ,XIO(Cfg_LSFail) XIO(Wrk_OpenFdbk) XIO(Wrk_ClosedFdbk) ] OTE(Sts_LSFail) MOV(3,Val_Fdbk) ,XIC(Wrk_OpenFdbk) XIO(Wrk_ClosedFdbk) MOV(2,Val_Fdbk) ,XIC(Wrk_ClosedFdbk) XIO(Wrk_OpenFdbk) OTE(Sts_Active) MOV(1,Val_Fdbk) ,[XIC(Cfg_LSFail) XIO(Wrk_OpenFdbk) XIO(Wrk_ClosedFdbk) ,XIO(Cfg_LSFail) XIC(Wrk_OpenFdbk) XIC(Wrk_ClosedFdbk) ] CLR(Val_Fdbk) ];
   // The rate limiter's scan timer must run and clear every scan, whether the Instruction
   // is true or not.  Doing so here avoids a bump in the Value on transition to EnableIn TRUE.
   14: TON(Wrk_ScanT,?,?)CLR(Wrk_ScanT.ACC);
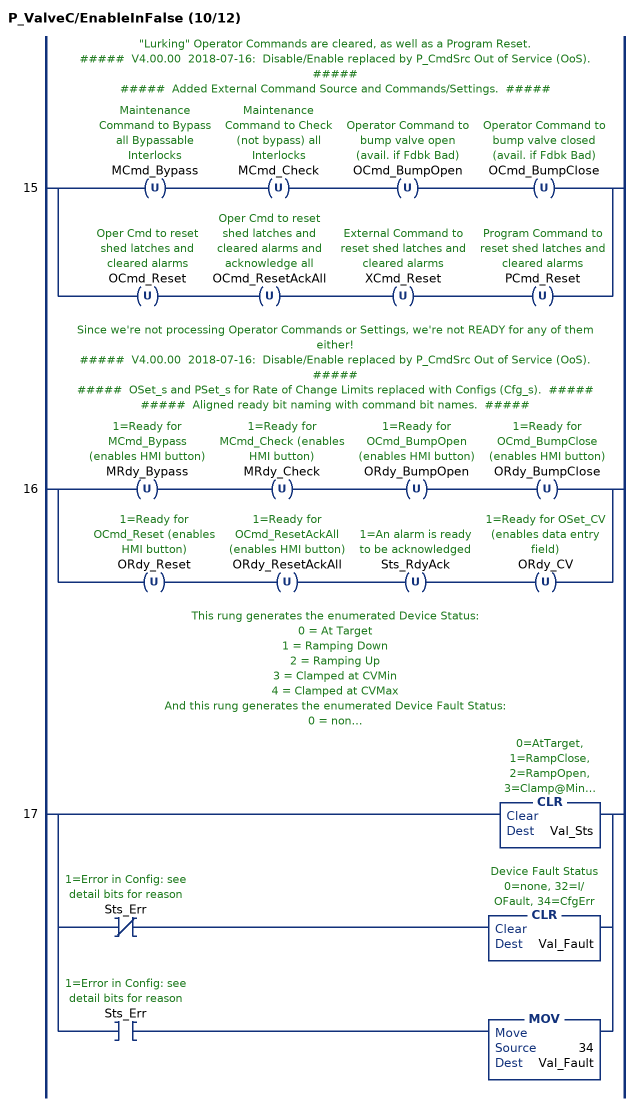
   // "Lurking" Operator Commands are cleared, as well as a Program Reset.
   // #####  V4.00.00  2018-07-16:  Disable/Enable replaced by P_CmdSrc Out of Service (OoS).  #####
   // #####  Added External Command Source and Commands/Settings.  #####
   15: [OTU(MCmd_Bypass) OTU(MCmd_Check) OTU(OCmd_BumpOpen) OTU(OCmd_BumpClose) ,OTU(OCmd_Reset) OTU(OCmd_ResetAckAll) OTU(XCmd_Reset) OTU(PCmd_Reset) ];
   // Since we're not processing Operator Commands or Settings, we're not READY for any of them either!
   // #####  V4.00.00  2018-07-16:  Disable/Enable replaced by P_CmdSrc Out of Service (OoS).  #####
   // #####  OSet_s and PSet_s for Rate of Change Limits replaced with Configs (Cfg_s).  #####
   // #####  Aligned ready bit naming with command bit names.  #####
   16: [OTU(MRdy_Bypass) OTU(MRdy_Check) OTU(ORdy_BumpOpen) OTU(ORdy_BumpClose) ,OTU(ORdy_Reset) OTU(ORdy_ResetAckAll) OTU(Sts_RdyAck) OTU(ORdy_CV) ];
   // This rung generates the enumerated Device Status:
   // 0 = At Target
   // 1 = Ramping Down
   // 2 = Ramping Up
   // 3 = Clamped at CVMin
   // 4 = Clamped at CVMax
   // And this rung generates the enumerated Device Fault Status:
   // 0 = none
   // 32 = I/O Fault
   // 34 = Configuration Error
   17: [CLR(Val_Sts) ,XIO(Sts_Err) CLR(Val_Fault) ,XIC(Sts_Err) MOV(34,Val_Fault) ];
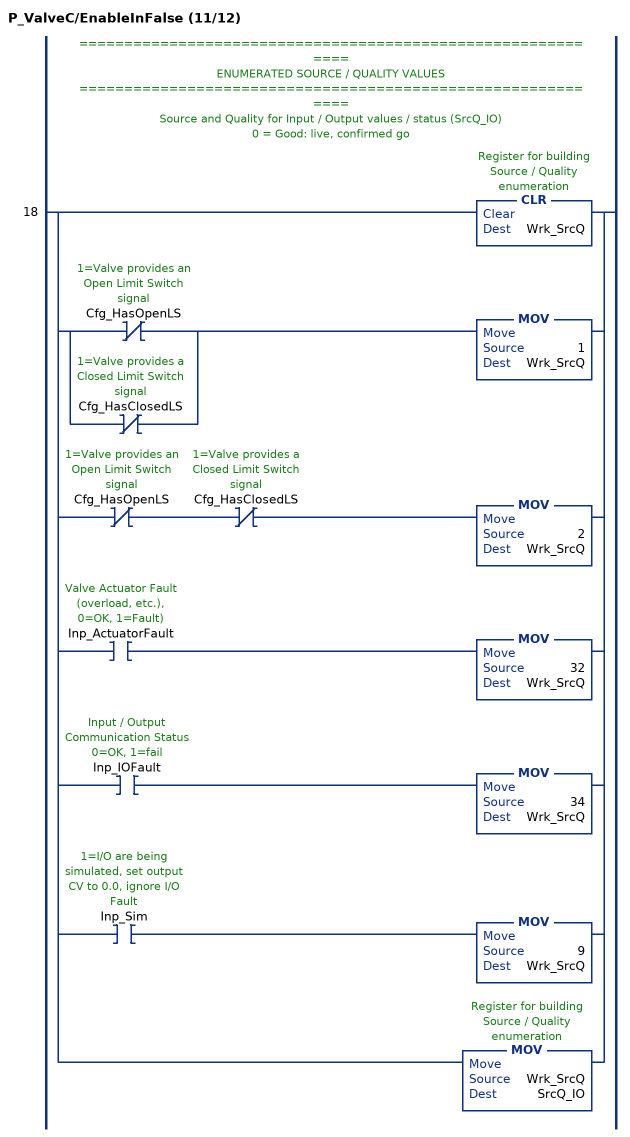
   // ============================================================
   // ENUMERATED SOURCE / QUALITY VALUES
   // ============================================================
   // Source and Quality for Input / Output values / status (SrcQ_IO)
   // 0 = Good: live, confirmed go
   18: [CLR(Wrk_SrcQ) ,[XIO(Cfg_HasOpenLS) ,XIO(Cfg_HasClosedLS) ] MOV(1,Wrk_SrcQ) ,XIO(Cfg_HasOpenLS) XIO(Cfg_HasClosedLS) MOV(2,Wrk_SrcQ) ,XIC(Inp_ActuatorFault) MOV(32,Wrk_SrcQ) ,XIC(Inp_IOFault) MOV(34,Wrk_SrcQ) ,XIC(Inp_Sim) MOV(9,Wrk_SrcQ) ,MOV(Wrk_SrcQ,SrcQ_IO) ];
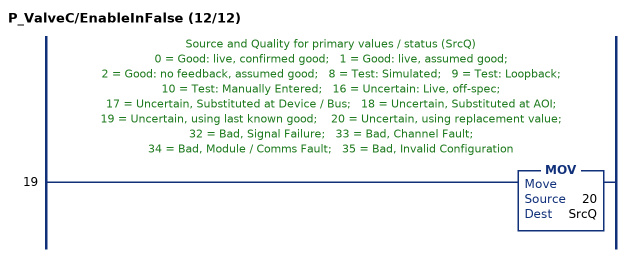
   // Source and Quality for primary values / status (SrcQ)
   // 0 = Good: live, confirmed good;   1 = Good: live, assumed good;
   // 2 = Good: no feedback, assumed good;   8 = Test: Simulated;   9 = Test: Loopback;
   // 10 = Test: Manually Entered;   16 = Uncertain: Live, off-spec;
   // 17 = Uncertain, Substituted at Device / Bus;   18 = Uncertain, Substituted at AOI;
   // 19 = Uncertain, using last known good;    20 = Uncertain, using replacement value;
   // 32 = Bad, Signal Failure;   33 = Bad, Channel Fault;
   // 34 = Bad, Module / Comms Fault;   35 = Bad, Invalid Configuration
   19: MOV(20,SrcQ);
END_ROUTINE

ROUTINE Logic   (* ladder *)
// Normal Scan: manipulate Control Valve with position feedback
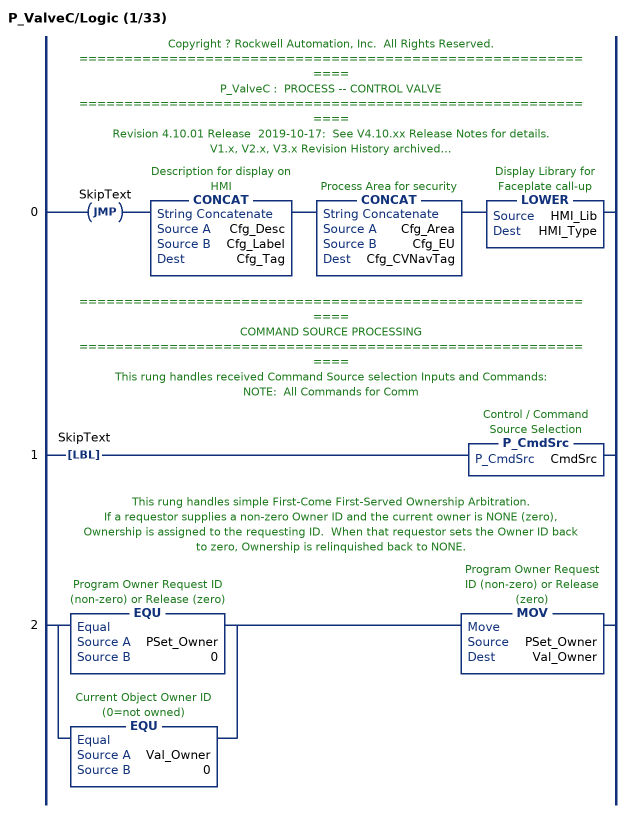
   // Copyright ? Rockwell Automation, Inc.  All Rights Reserved.
   // ============================================================
   // P_ValveC :  PROCESS -- CONTROL VALVE
   // ============================================================
   // Revision 4.10.01 Release  2019-10-17:  See V4.10.xx Release Notes for details.
   // V1.x, V2.x, V3.x Revision History archived.
   // V4.00.00  2018-07-16:  Changed Inf_ items to HMI_, and added Cfg_Area for security.
   // Added notify and unack count rollup for associated object(s).
   // Changed "Mode" to "Command Source" using P_CmdSrc 4.00.00.
   // Deleted Cfg_PCmdClear; all Program Commands are now self-clearing.
   // Aligned ready bit naming with command bit names.
   // Added unacked alarm count.
   // Added configurable decimal places for display on HMI.
   // All OCmds/MCmds and ORdys/MRdys are now Local Tags.
   // Added Sts_RdyAck and Sts_RdyReset for use by external objects.
   // Added option for no position feedback (simulated with hysteresis).
   // V4.10.00  2019-03-08:  Added option to clamp to a full/empty range when we have
   // limit switches. Changed availability to use input availability from interlocks.
   // Updated to P_CmdSrc V4.10.00. Corrected parameter External Access.
   // Added Cfg_HasMoreObj.
   // V4.10.01  2019-10-17:  No changes, uprevved because P_CmdSrc 4.10.01 is used.
   // ============================================================
   // This Instruction controls an Analog or Pulse Output Valve with
   // analog or simulated position feedback and provides:
   // *  Program and Operator entry of target position in Percent Open
   // *  Ramping of position to target at specified Rate of Change (%/sec)
   // *  Scaling of Position Feedback input from Raw (I/O card) Units to percent
   // *  Monitoring of Interlock conditions which cause output to shed
   // *  Configurable shed to HOLD or to configured position
   // *  Monitoring of I/O communication faults
   // *  Alarms for Interlock Trip, Actuator Fault, I/O Fault
   // *  Opened, Closed status based on limit switches (if provided),
   // or based on Position Feedback and a configured threshold.
   // *  "Available" status for use by automation logic to know whether valve
   //       can be controlled by other objects.
   // Command Sources are arbitrated by a P_CmdSrc Add-On Instruction instance.
   // Command Sources: Operator, Program, External, Override, Maintenance, Out of Service, Hand.
   // Alarms are provided by P_Alarm Add-On Instruction instances.
   // ============================================================
   // SHOW LOCAL STRINGS
   // ============================================================
   // The STRINGs containing the text associated with each instance of this
   // instruction cannot be Input or Output Parameters, because STRINGs are not
   //  'atomic' types. (Inputs and Outputs must be SINT, INT, DINT, REAL, or BOOL.)
   // In order to make it easier to find and configure these STRINGs, this rung
   // was added.  THE JMP (and the LBL on the following rung)
   // MUST NOT BE REMOVED!!!
   // To view the STRINGs, go to the instruction instance (in LD or FBD), RIGHT-click
   // to bring up the context menu and select "Open Instruction Logic".
   // This rung will appear with the STRING values for the selected instance.
   // You may double-click the STRING values here to modify them as well.
   // #####  V4.00.00  2018-07-16:  Added string for Cfg_Area, renamed Inf_* to HMI_*.  #####
   0: JMP(SkipText)CONCAT(Cfg_Desc,Cfg_Label,Cfg_Tag)CONCAT(Cfg_Area,Cfg_EU,Cfg_CVNavTag)LOWER(HMI_Lib,HMI_Type);
   // ============================================================
   // COMMAND SOURCE PROCESSING
   // ============================================================
   // This rung handles received Command Source selection Inputs and Commands:
   // NOTE:  All Commands for Comm
   1: LBL(SkipText)P_CmdSrc(CmdSrc);
   // This rung handles simple First-Come First-Served Ownership Arbitration.
   // If a requestor supplies a non-zero Owner ID and the current owner is NONE (zero),
   // Ownership is assigned to the requesting ID.  When that requestor sets the Owner ID back
   // to zero, Ownership is relinquished back to NONE.
   2: [EQU(PSet_Owner,0) ,EQU(Val_Owner,0) ]MOV(PSet_Owner,Val_Owner);
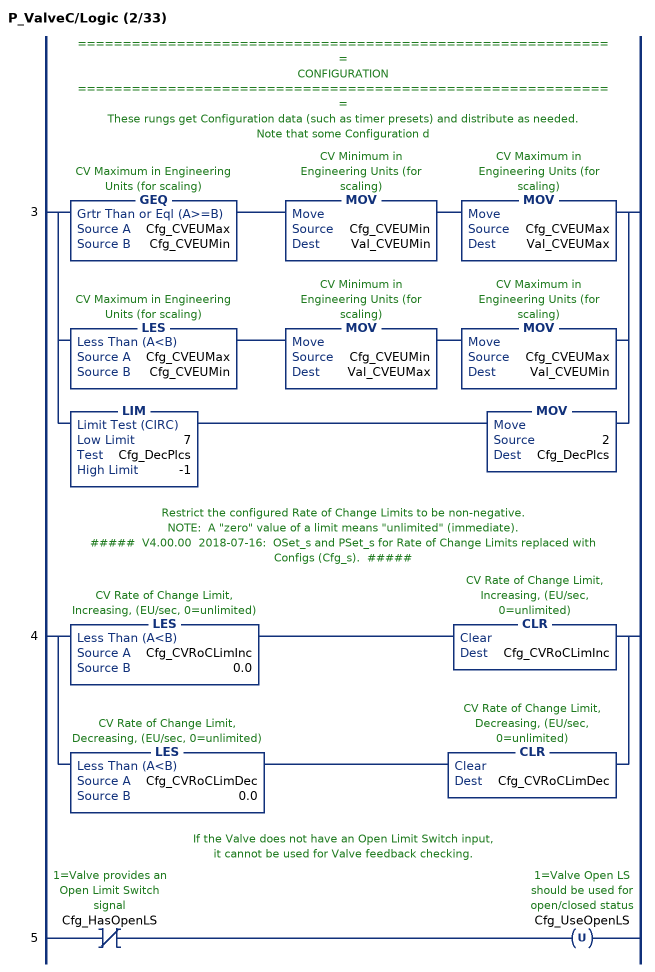
   // ============================================================
   // CONFIGURATION
   // ============================================================
   // These rungs get Configuration data (such as timer presets) and distribute as needed.
   // Note that some Configuration d
   3: [GEQ(Cfg_CVEUMax,Cfg_CVEUMin) MOV(Cfg_CVEUMin,Val_CVEUMin) MOV(Cfg_CVEUMax,Val_CVEUMax) ,LES(Cfg_CVEUMax,Cfg_CVEUMin) MOV(Cfg_CVEUMin,Val_CVEUMax) MOV(Cfg_CVEUMax,Val_CVEUMin) ,LIM(7,Cfg_DecPlcs,-1) MOV(2,Cfg_DecPlcs) ];
   // Restrict the configured Rate of Change Limits to be non-negative.
   // NOTE:  A "zero" value of a limit means "unlimited" (immediate).
   // #####  V4.00.00  2018-07-16:  OSet_s and PSet_s for Rate of Change Limits replaced with Configs (Cfg_s).  #####
   4: [LES(Cfg_CVRoCLimInc,0.0) CLR(Cfg_CVRoCLimInc) ,LES(Cfg_CVRoCLimDec,0.0) CLR(Cfg_CVRoCLimDec) ];
   // If the Valve does not have an Open Limit Switch input,
   // it cannot be used for Valve feedback checking.
   5: XIO(Cfg_HasOpenLS)OTU(Cfg_UseOpenLS);
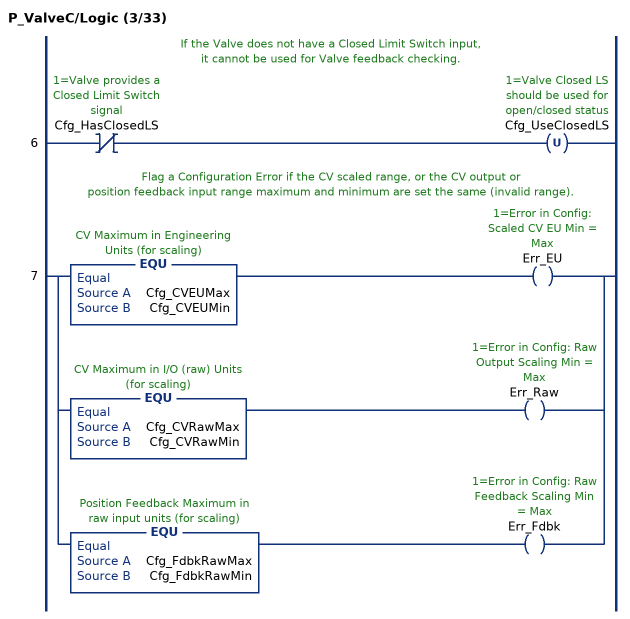
   // If the Valve does not have a Closed Limit Switch input,
   // it cannot be used for Valve feedback checking.
   6: XIO(Cfg_HasClosedLS)OTU(Cfg_UseClosedLS);
   // Flag a Configuration Error if the CV scaled range, or the CV output or
   // position feedback input range maximum and minimum are set the same (invalid range).
   7: [EQU(Cfg_CVEUMax,Cfg_CVEUMin) OTE(Err_EU) ,EQU(Cfg_CVRawMax,Cfg_CVRawMin) OTE(Err_Raw) ,EQU(Cfg_FdbkRawMax,Cfg_FdbkRawMin) OTE(Err_Fdbk) ];
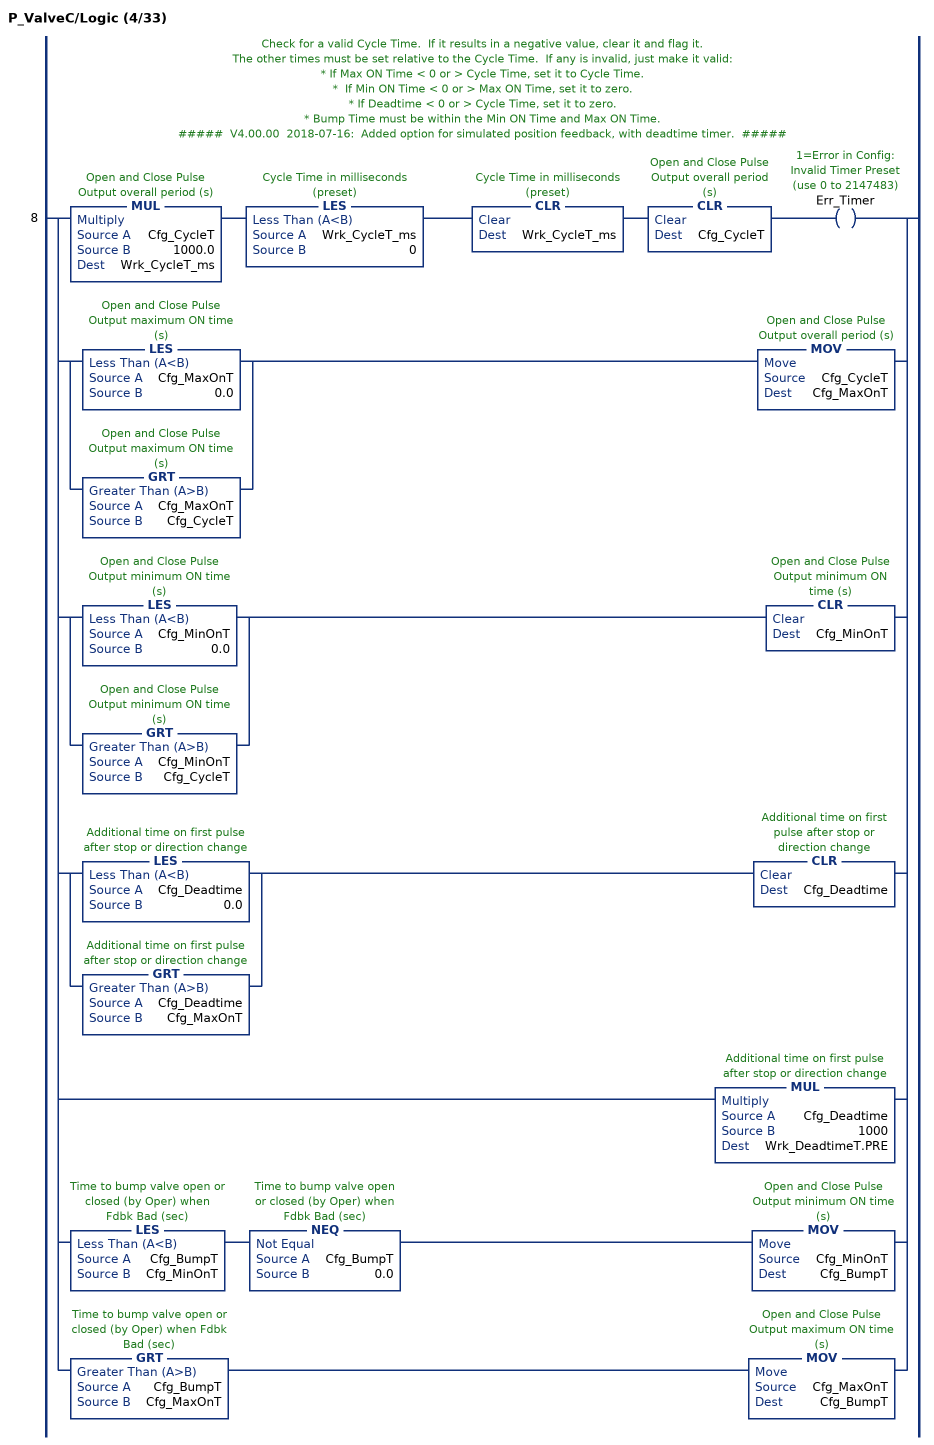
   // Check for a valid Cycle Time.  If it results in a negative value, clear it and flag it.
   // The other times must be set relative to the Cycle Time.  If any is invalid, just make it valid:
   // * If Max ON Time < 0 or > Cycle Time, set it to Cycle Time.
   // *  If Min ON Time < 0 or > Max ON Time, set it to zero.
   // * If Deadtime < 0 or > Cycle Time, set it to zero.
   // * Bump Time must be within the Min ON Time and Max ON Time.
   // #####  V4.00.00  2018-07-16:  Added option for simulated position feedback, with deadtime timer.  #####
   8: [MUL(Cfg_CycleT,1000.0,Wrk_CycleT_ms) LES(Wrk_CycleT_ms,0) CLR(Wrk_CycleT_ms) CLR(Cfg_CycleT) OTE(Err_Timer) ,[LES(Cfg_MaxOnT,0.0) ,GRT(Cfg_MaxOnT,Cfg_CycleT) ] MOV(Cfg_CycleT,Cfg_MaxOnT) ,[LES(Cfg_MinOnT,0.0) ,GRT(Cfg_MinOnT,Cfg_CycleT) ] CLR(Cfg_MinOnT) ,[LES(Cfg_Deadtime,0.0) ,GRT(Cfg_Deadtime,Cfg_MaxOnT) ] CLR(Cfg_Deadtime) ,MUL(Cfg_Deadtime,1000,Wrk_DeadtimeT.PRE) ,LES(Cfg_BumpT,Cfg_MinOnT) NEQ(Cfg_BumpT,0.0) MOV(Cfg_MinOnT,Cfg_BumpT) ,GRT(Cfg_BumpT,Cfg_MaxOnT) MOV(Cfg_MaxOnT,Cfg_BumpT) ];
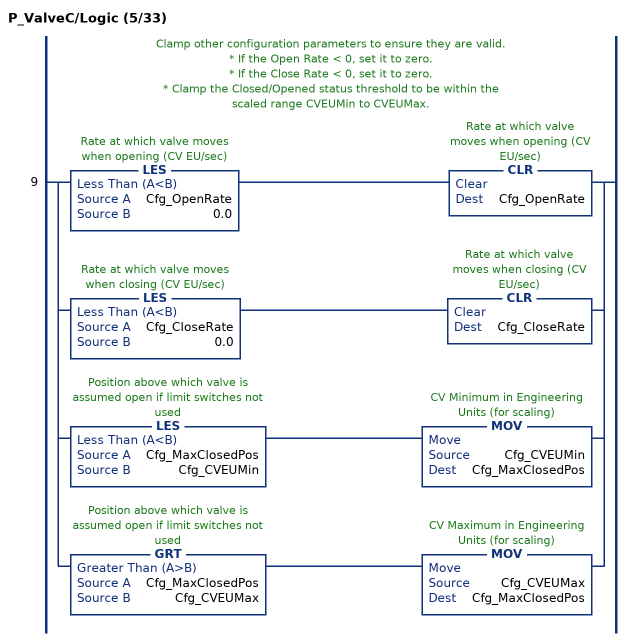
   // Clamp other configuration parameters to ensure they are valid.
   // * If the Open Rate < 0, set it to zero.
   // * If the Close Rate < 0, set it to zero.
   // * Clamp the Closed/Opened status threshold to be within the
   // scaled range CVEUMin to CVEUMax.
   9: [LES(Cfg_OpenRate,0.0) CLR(Cfg_OpenRate) ,LES(Cfg_CloseRate,0.0) CLR(Cfg_CloseRate) ,LES(Cfg_MaxClosedPos,Cfg_CVEUMin) MOV(Cfg_CVEUMin,Cfg_MaxClosedPos) ,GRT(Cfg_MaxClosedPos,Cfg_CVEUMax) MOV(Cfg_CVEUMax,Cfg_MaxClosedPos) ];
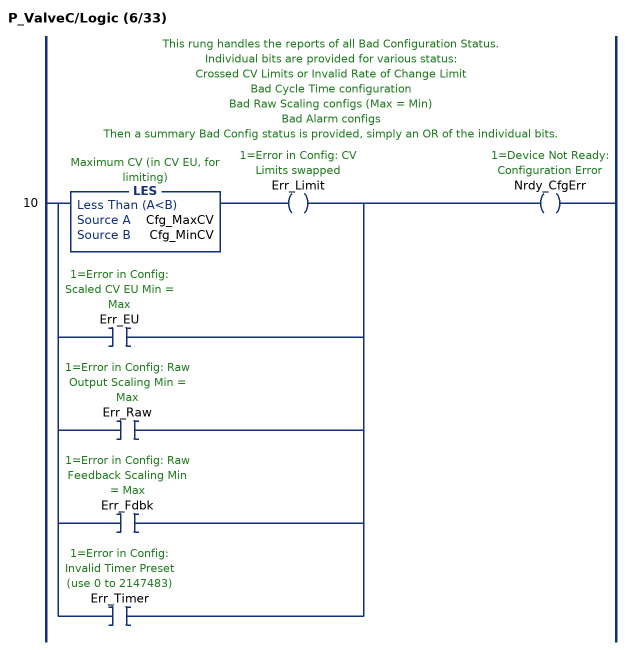
   // This rung handles the reports of all Bad Configuration Status.
   // Individual bits are provided for various status:
   // Crossed CV Limits or Invalid Rate of Change Limit
   // Bad Cycle Time configuration
   // Bad Raw Scaling configs (Max = Min)
   // Bad Alarm configs
   // Then a summary Bad Config status is provided, simply an OR of the individual bits.
   10: [LES(Cfg_MaxCV,Cfg_MinCV) OTE(Err_Limit) ,XIC(Err_EU) ,XIC(Err_Raw) ,XIC(Err_Fdbk) ,XIC(Err_Timer) ]OTE(Nrdy_CfgErr);
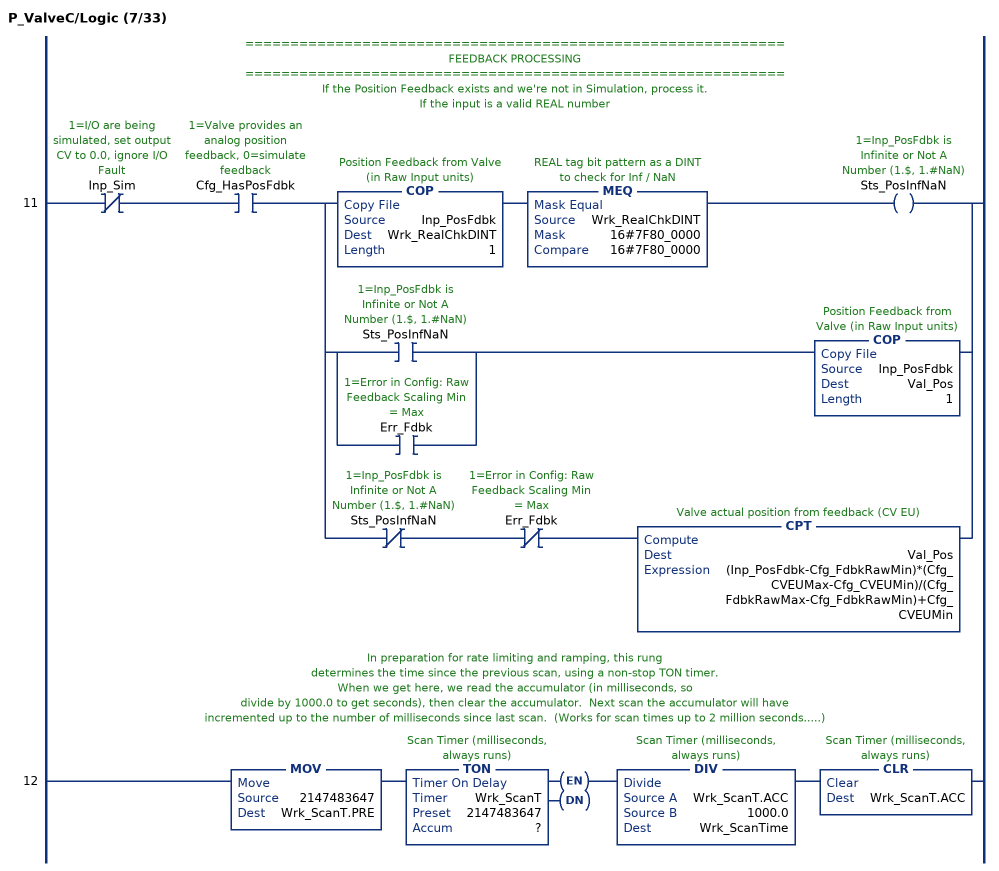
   // ============================================================
   // FEEDBACK PROCESSING
   // ============================================================
   // If the Position Feedback exists and we're not in Simulation, process it.
   // If the input is a valid REAL number
   11: XIO(Inp_Sim)XIC(Cfg_HasPosFdbk)[COP(Inp_PosFdbk,Wrk_RealChkDINT,1) MEQ(Wrk_RealChkDINT,16#7F80_0000,16#7F80_0000) OTE(Sts_PosInfNaN) ,[XIC(Sts_PosInfNaN) ,XIC(Err_Fdbk) ] COP(Inp_PosFdbk,Val_Pos,1) ,XIO(Sts_PosInfNaN) XIO(Err_Fdbk) CPT(Val_Pos,(Inp_PosFdbk-Cfg_FdbkRawMin)*(Cfg_CVEUMax-Cfg_CVEUMin)/(Cfg_FdbkRawMax-Cfg_FdbkRawMin)+Cfg_CVEUMin) ];
   // In preparation for rate limiting and ramping, this rung
   // determines the time since the previous scan, using a non-stop TON timer.
   // When we get here, we read the accumulator (in milliseconds, so
   // divide by 1000.0 to get seconds), then clear the accumulator.  Next scan the accumulator will have
   // incremented up to the number of milliseconds since last scan.  (Works for scan times up to 2 million seconds.....)
   12: MOV(2147483647,Wrk_ScanT.PRE)TON(Wrk_ScanT,?,?)DIV(Wrk_ScanT.ACC,1000.0,Wrk_ScanTime)CLR(Wrk_ScanT.ACC);
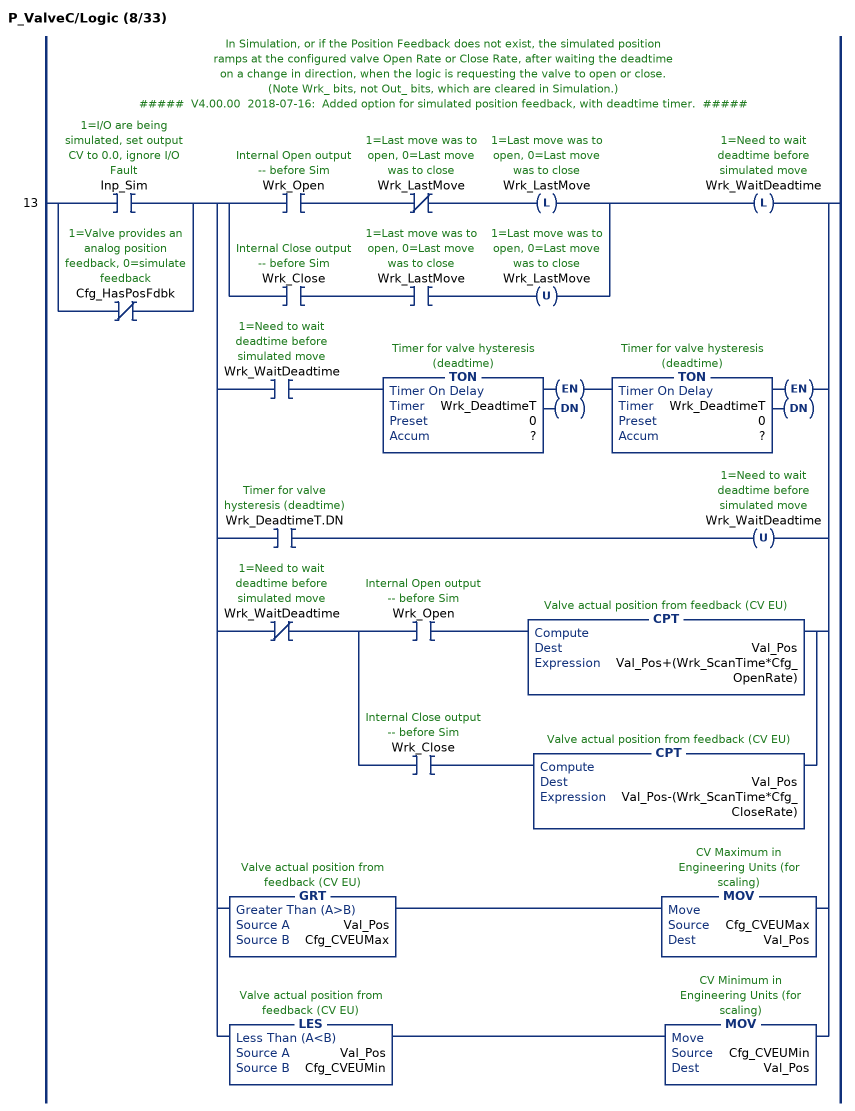
   // In Simulation, or if the Position Feedback does not exist, the simulated position
   // ramps at the configured valve Open Rate or Close Rate, after waiting the deadtime
   // on a change in direction, when the logic is requesting the valve to open or close.
   // (Note Wrk_ bits, not Out_ bits, which are cleared in Simulation.)
   // #####  V4.00.00  2018-07-16:  Added option for simulated position feedback, with deadtime timer.  #####
   13: [XIC(Inp_Sim) ,XIO(Cfg_HasPosFdbk) ][[XIC(Wrk_Open) XIO(Wrk_LastMove) OTL(Wrk_LastMove) ,XIC(Wrk_Close) XIC(Wrk_LastMove) OTU(Wrk_LastMove) ] OTL(Wrk_WaitDeadtime) ,XIC(Wrk_WaitDeadtime) TON(Wrk_DeadtimeT,?,?) TON(Wrk_DeadtimeT,?,?) ,XIC(Wrk_DeadtimeT.DN) OTU(Wrk_WaitDeadtime) ,XIO(Wrk_WaitDeadtime) [XIC(Wrk_Open) CPT(Val_Pos,Val_Pos+(Wrk_ScanTime*Cfg_OpenRate)) ,XIC(Wrk_Close) CPT(Val_Pos,Val_Pos-(Wrk_ScanTime*Cfg_CloseRate)) ] ,GRT(Val_Pos,Cfg_CVEUMax) MOV(Cfg_CVEUMax,Val_Pos) ,LES(Val_Pos,Cfg_CVEUMin) MOV(Cfg_CVEUMin,Val_Pos) ];
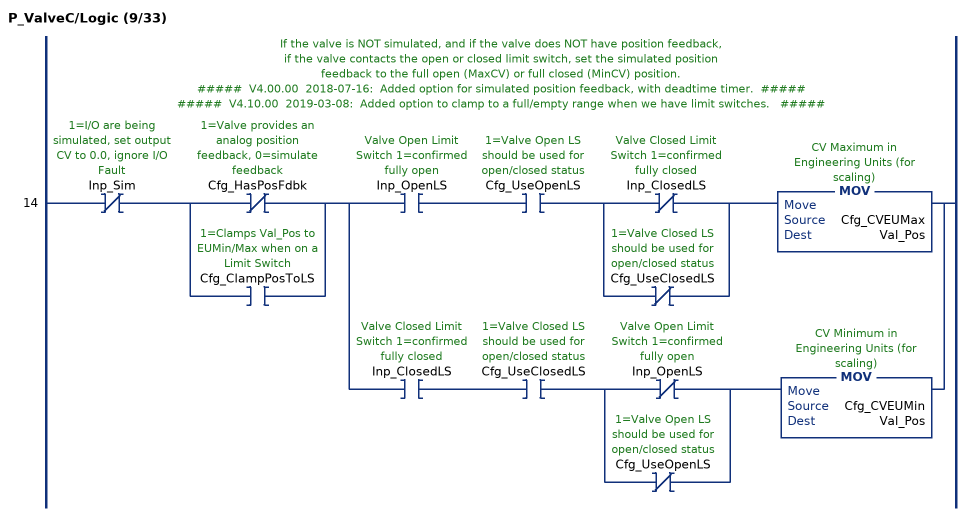
   // If the valve is NOT simulated, and if the valve does NOT have position feedback,
   // if the valve contacts the open or closed limit switch, set the simulated position
   // feedback to the full open (MaxCV) or full closed (MinCV) position.
   // #####  V4.00.00  2018-07-16:  Added option for simulated position feedback, with deadtime timer.  #####
   // #####  V4.10.00  2019-03-08:  Added option to clamp to a full/empty range when we have limit switches.   #####
   14: XIO(Inp_Sim)[XIO(Cfg_HasPosFdbk) ,XIC(Cfg_ClampPosToLS) ][XIC(Inp_OpenLS) XIC(Cfg_UseOpenLS) [XIO(Inp_ClosedLS) ,XIO(Cfg_UseClosedLS) ] MOV(Cfg_CVEUMax,Val_Pos) ,XIC(Inp_ClosedLS) XIC(Cfg_UseClosedLS) [XIO(Inp_OpenLS) ,XIO(Cfg_UseOpenLS) ] MOV(Cfg_CVEUMin,Val_Pos) ];
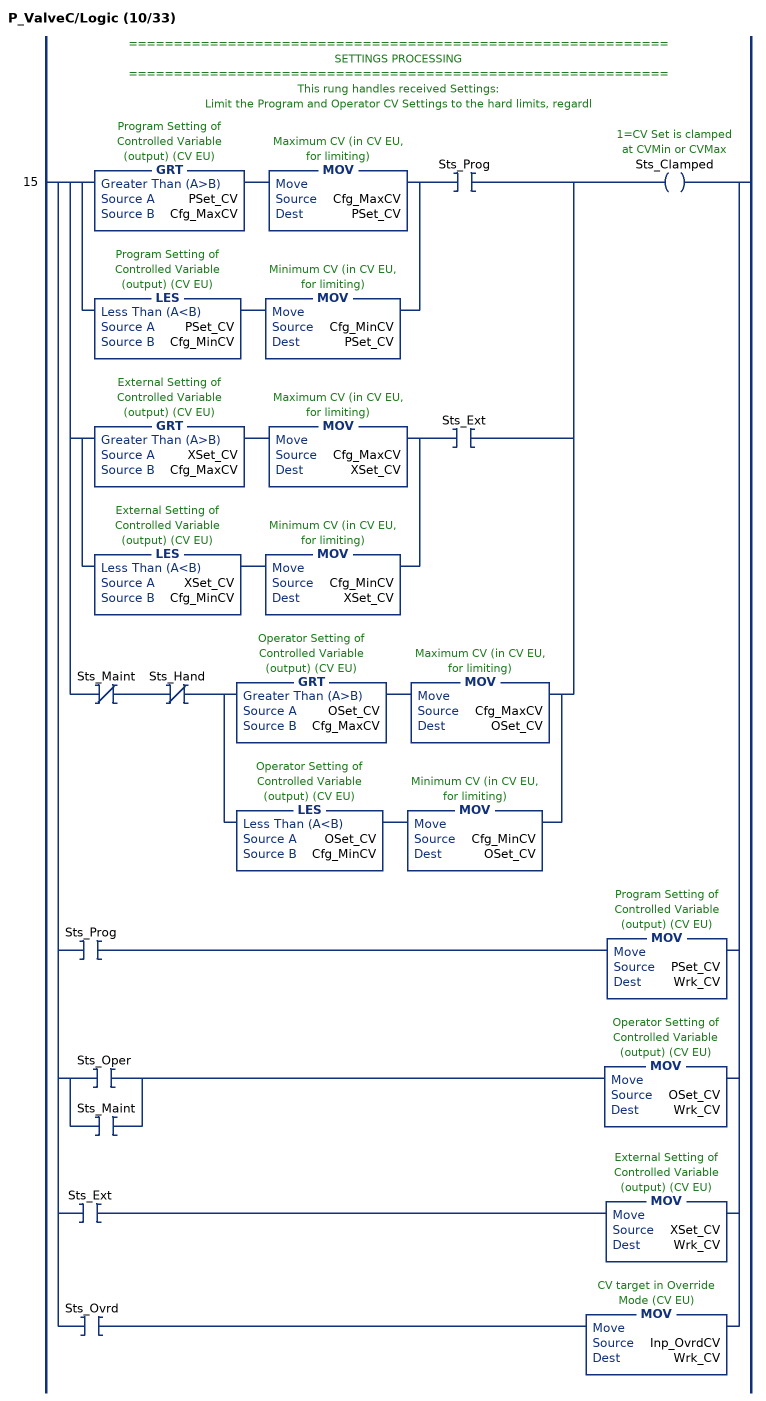
   // ============================================================
   // SETTINGS PROCESSING
   // ============================================================
   // This rung handles received Settings:
   // Limit the Program and Operator CV Settings to the hard limits, regardl
   15: [[[GRT(PSet_CV,Cfg_MaxCV) MOV(Cfg_MaxCV,PSet_CV) ,LES(PSet_CV,Cfg_MinCV) MOV(Cfg_MinCV,PSet_CV) ] XIC(Sts_Prog) ,[GRT(XSet_CV,Cfg_MaxCV) MOV(Cfg_MaxCV,XSet_CV) ,LES(XSet_CV,Cfg_MinCV) MOV(Cfg_MinCV,XSet_CV) ] XIC(Sts_Ext) ,XIO(Sts_Maint) XIO(Sts_Hand) [GRT(OSet_CV,Cfg_MaxCV) MOV(Cfg_MaxCV,OSet_CV) ,LES(OSet_CV,Cfg_MinCV) MOV(Cfg_MinCV,OSet_CV) ] ] OTE(Sts_Clamped) ,XIC(Sts_Prog) MOV(PSet_CV,Wrk_CV) ,[XIC(Sts_Oper) ,XIC(Sts_Maint) ] MOV(OSet_CV,Wrk_CV) ,XIC(Sts_Ext) MOV(XSet_CV,Wrk_CV) ,XIC(Sts_Ovrd) MOV(Inp_OvrdCV,Wrk_CV) ];
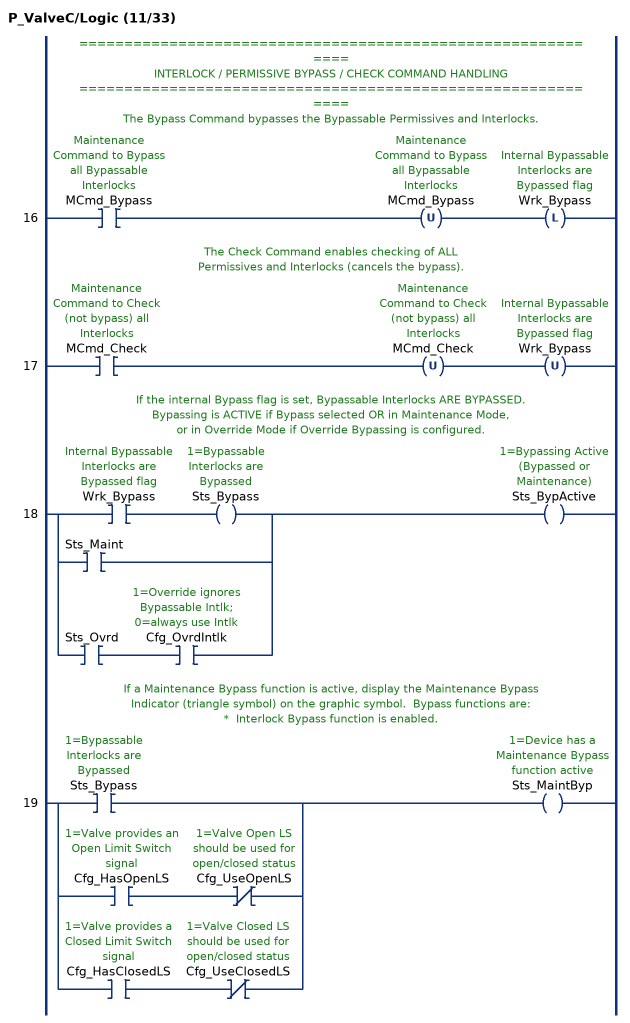
   // ============================================================
   // INTERLOCK / PERMISSIVE BYPASS / CHECK COMMAND HANDLING
   // ============================================================
   // The Bypass Command bypasses the Bypassable Permissives and Interlocks.
   16: XIC(MCmd_Bypass)OTU(MCmd_Bypass)OTL(Wrk_Bypass);
   // The Check Command enables checking of ALL
   // Permissives and Interlocks (cancels the bypass).
   17: XIC(MCmd_Check)OTU(MCmd_Check)OTU(Wrk_Bypass);
   // If the internal Bypass flag is set, Bypassable Interlocks ARE BYPASSED.
   // Bypassing is ACTIVE if Bypass selected OR in Maintenance Mode,
   // or in Override Mode if Override Bypassing is configured.
   18: [XIC(Wrk_Bypass) OTE(Sts_Bypass) ,XIC(Sts_Maint) ,XIC(Sts_Ovrd) XIC(Cfg_OvrdIntlk) ]OTE(Sts_BypActive);
   // If a Maintenance Bypass function is active, display the Maintenance Bypass
   // Indicator (triangle symbol) on the graphic symbol.  Bypass functions are:
   // *  Interlock Bypass function is enabled.
   19: [XIC(Sts_Bypass) ,XIC(Cfg_HasOpenLS) XIO(Cfg_UseOpenLS) ,XIC(Cfg_HasClosedLS) XIO(Cfg_UseClosedLS) ]OTE(Sts_MaintByp);
